      L     L#0;
      U     "MAL1S033Par".Par.FlagProcess.ProcessActive;
      SPBN  n609; // no addition
      SET   ;
      S     "MAL1S033Par".Par.FlagProcess.Inf21; // add heat quantity
      U     "SYS_Scan0_Tick1s"; // scan 1sec
      SPBN  E609;
      L     "MAL1S033Par".Par.ProcessValue_Real.Value05; // heat quantity in kW
      +R    ;
      T     "MAL1S033Par".Par.ProcessValue_Real.Value05;
      SPA   E609;
n609: NOP   0;
      U     "MAL1S033Par".Par.FlagProcess.Inf21; // add heat quantity
      SPBN  E609;
      R     "MAL1S033Par".Par.FlagProcess.Inf21; // add heat quantity
      L     "MAL1S033Par".Par.ProcessValue_Real.Value05;
      L     3.600000e+003;
      /R    ; // from kWs to kWh
      L     1.000000e+003;
      /R    ; // from kWh to MWh
      RND   ;
      T     "MAL1S033Par".Par.ProcessValue_Real.Value06; // result to batch potokoll
      L     0.000000e+000; // clear calculator
      T     "MAL1S033Par".Par.ProcessValue_Real.Value05;
E609: NOP   0;
NETWORK
TITLE =ASW_7000: Step loading kilning
//
      U     "MAL1S033".ToASW.InfDataReady;
      U     "MAL1S033".PCRead.Step.StWait;
      U     "MAL1S033".PCWrite.ExtFuncOn.StartLoading; // PIC command "start loading"
      S     "MAL1S033Par".Par.FlagFunction_1.StepLoading; // Step loading
      R     "MAL1S033Par".Par.FlagMachine.ImpulsNullstellung;
      R     "MAL1S033Par".Par.FlagMachine.CmdTurnRevAfterLoading;
      R     "MAL1S033Par".Par.FlagMachine.CmdTurnFwdAfterLoading;
//
      SET   ;
      R     "MAL1S033".PCWrite.ExtFuncOn.StartLoading; // PIC command "start loading"
//
      U     "MAL1S033".ToASW.InfDataReady;
      U     "MAL1S033".PCRead.Step.StActive;
      U     "MAL1S033Par".Par.FlagFunction_1.StepLoading; // Step loading
      SPB   e71;
      R     "MAL1S033Par".Par.Switches1.StaOn00; // LiftingPositionRound_1
      R     "MAL1S033Par".Par.Switches1.StaOn01; // LiftingPositionRound_2
      R     "MAL1S033Par".Par.Switches1.StaOn02; // LiftingPositionRound_3
      R     "MAL1S033Par".Par.Switches1.StaOn03; // LiftingPositionRound_4
      R     "MAL1S033Par".Par.Switches1.StaOn04; // LiftingPositionRound_5
      R     "MAL1S033Par".Par.Switches1.StaOn05; // LiftingPositionRound_6
e71:  NOP   0;
      U     "MAL1S033".ToASW.InfDataReady;
      U     "MAL1S033".PCRead.Step.StActive;
      U     "MAL1S033Par".Par.FlagFunction_1.StepLoading; // Step loading
      UN    "MAL1S033Par".Par.FlagFunction_1.FinishLoading;
      UN    "MAL1S033Par".Par.FlagFunction_1.LoadEnd;
      SPBN  E700;
      U(    ;
      U(    ;
      L     "G292M".A_3211_MXZ41MA.Ma.OutPositionAngle;
      L     3460; // 346.0°
      >=I   ;
      )     ;
      O     ;
      U(    ;
      L     "G292M".A_3211_MXZ41MA.Ma.OutCntRound;
      L     L#1;
      >=D   ;
      )     ;
      )     ;
      U     "MAL1S033Par".Par.FlagFunction_1.StepLoading;
      =     "MAL1S033Par".Par.FlagFunction_0.ReducedSpeed;
//
      L     "MAL1S033Par".RecipeHeader.Loading.LiftingPositionRound_3;
      L     20; // 20°
      -I    ;
      T     "MAL1S033Par".Par.ParIntMachine.LiftingPositionRound_4;
      L     "MAL1S033Par".RecipeHeader.Loading.LoadingLevelRound_3;
      L     "MAL1S033Par".RecipeHeader.Loading.OffsetLevelNextRound;
      +I    ;
      T     "MAL1S033Par".Par.ParIntMachine.LoadingLevelRound_4;
//
      L     "MAL1S033Par".Par.ParIntMachine.LiftingPositionRound_4;
      L     20; // 20°
      -I    ;
      T     "MAL1S033Par".Par.ParIntMachine.LiftingPositionRound_5;
      L     "MAL1S033Par".Par.ParIntMachine.LoadingLevelRound_4;
      L     "MAL1S033Par".RecipeHeader.Loading.OffsetLevelNextRound;
      +I    ;
      T     "MAL1S033Par".Par.ParIntMachine.LoadingLevelRound_5;
//
      L     "MAL1S033Par".Par.ParIntMachine.LiftingPositionRound_5;
      L     20; // 20°
      -I    ;
      T     "MAL1S033Par".Par.ParIntMachine.LiftingPositionRound_6;
      L     "MAL1S033Par".Par.ParIntMachine.LoadingLevelRound_5;
      L     "MAL1S033Par".RecipeHeader.Loading.OffsetLevelNextRound;
      +I    ;
      T     "MAL1S033Par".Par.ParIntMachine.LoadingLevelRound_6;
//
      L     3600;
      L     "G292M".A_3211_MXZ41MA.Ma.Par.ParTolPosition;
      -I    ;
      L     "G292M".A_3211_MXZ41MA.Ma.OutPositionAngle;
      <=I   ;
      SPB   E700;
//
      L     "G292M".A_3211_MXZ41MA.Ma.OutPositionAngle;
      L     0;
      <I    ;
//      <=I
      SPB   E700;
//
      L     "G292M".A_3211_MXZ41MA.Ma.OutPositionAngle;
      L     10;
      /I    ;
      T     "MAL1S033Par".Par.MachineValue.ISTWERT_FAHRANTRIEB_POSI;
//
      U     "MAL1S033Par".Par.FlagFunction_1.StepLoading; // Step loading
      FP    "MAL1S033Par".Par.Switches1.StaOn08;
      =     "MAL1S033Par".Par.Switches1.StaOn09; // scan start loading
      U     "MAL1S033Par".Par.Switches1.StaOn09; // scan start loading
      SPBN  e72;
      R     "MAL1S033Par".Par.Switches1.StaOn00; // LiftingPositionRound_1
      R     "MAL1S033Par".Par.Switches1.StaOn01; // LiftingPositionRound_2
      R     "MAL1S033Par".Par.Switches1.StaOn02; // LiftingPositionRound_3
      R     "MAL1S033Par".Par.Switches1.StaOn03; // LiftingPositionRound_4
      R     "MAL1S033Par".Par.Switches1.StaOn04; // LiftingPositionRound_5
      R     "MAL1S033Par".Par.Switches1.StaOn05; // LiftingPositionRound_6
//
e72:  NOP   0;
//
      U(    ;
      L     "G292M".A_3211_MXZ41MA.Ma.OutCntRound;
      L     L#0;
      ==D   ;
      )     ;
      U(    ;
      L     "MAL1S033Par".Par.MachineValue.ISTWERT_FAHRANTRIEB_POSI;
      L     "MAL1S033Par".RecipeHeader.Loading.LiftingPositionRound_1;
      <I    ;
      )     ;
      S     "MAL1S033Par".Par.Switches1.StaOn00; // LiftingPositionRound_1
//
      U(    ;
      L     "G292M".A_3211_MXZ41MA.Ma.OutCntRound;
      L     L#0;
      ==D   ;
      )     ;
      U(    ;
      L     "MAL1S033Par".Par.MachineValue.ISTWERT_FAHRANTRIEB_POSI;
      L     "MAL1S033Par".RecipeHeader.Loading.LiftingPositionRound_1;
      >=I   ;
      )     ;
      U(    ;
      L     "MAL1S033Par".Par.MachineValue.ISTWERT_FAHRANTRIEB_POSI;
      L     3550; // 355.0° --> Ruckeln am Nullpunkt abfangen
      <=I   ;
      )     ;
      S     "MAL1S033Par".Par.Switches1.StaOn01; // LiftingPositionRound_2
//
      U     "MAL1S033Par".Par.Switches1.StaOn01; // LiftingPositionRound_2
      R     "MAL1S033Par".Par.Switches1.StaOn00; // LiftingPositionRound_1
//
      U(    ;
      L     "G292M".A_3211_MXZ41MA.Ma.OutCntRound;
      L     L#1;
      ==D   ;
      )     ;
      U(    ;
      L     "MAL1S033Par".Par.MachineValue.ISTWERT_FAHRANTRIEB_POSI;
      L     "MAL1S033Par".RecipeHeader.Loading.LiftingPositionRound_2;
      >=I   ;
      )     ;
      S     "MAL1S033Par".Par.Switches1.StaOn02; // LiftingPositionRound_3
//
      U     "MAL1S033Par".Par.Switches1.StaOn02; // LiftingPositionRound_3
      R     "MAL1S033Par".Par.Switches1.StaOn01; // LiftingPositionRound_2
      R     "MAL1S033Par".Par.Switches1.StaOn00; // LiftingPositionRound_1
//
      U(    ;
      L     "G292M".A_3211_MXZ41MA.Ma.OutCntRound;
      L     L#2;
      ==D   ;
      )     ;
      U(    ;
      L     "MAL1S033Par".Par.MachineValue.ISTWERT_FAHRANTRIEB_POSI;
      L     "MAL1S033Par".RecipeHeader.Loading.LiftingPositionRound_3;
      >=I   ;
      )     ;
      S     "MAL1S033Par".Par.Switches1.StaOn03; // LiftingPositionRound_4
//
      U     "MAL1S033Par".Par.Switches1.StaOn03; // LiftingPositionRound_4
      R     "MAL1S033Par".Par.Switches1.StaOn02; // LiftingPositionRound_3
      R     "MAL1S033Par".Par.Switches1.StaOn01; // LiftingPositionRound_2
      R     "MAL1S033Par".Par.Switches1.StaOn00; // LiftingPositionRound_1
      U(    ;
      L     "G292M".A_3211_MXZ41MA.Ma.OutCntRound;
      L     L#3;
      ==D   ;
      )     ;
      U(    ;
      L     "MAL1S033Par".Par.MachineValue.ISTWERT_FAHRANTRIEB_POSI;
      L     "MAL1S033Par".Par.ParIntMachine.LiftingPositionRound_4;
      >=I   ;
      )     ;
      S     "MAL1S033Par".Par.Switches1.StaOn04; // LiftingPositionRound_5
//
      U     "MAL1S033Par".Par.Switches1.StaOn04; // LiftingPositionRound_5
      R     "MAL1S033Par".Par.Switches1.StaOn03; // LiftingPositionRound_4
      R     "MAL1S033Par".Par.Switches1.StaOn02; // LiftingPositionRound_3
      R     "MAL1S033Par".Par.Switches1.StaOn01; // LiftingPositionRound_2
      R     "MAL1S033Par".Par.Switches1.StaOn00; // LiftingPositionRound_1
      U(    ;
      L     "G292M".A_3211_MXZ41MA.Ma.OutCntRound;
      L     L#4;
      ==D   ;
      )     ;
      U(    ;
      L     "MAL1S033Par".Par.MachineValue.ISTWERT_FAHRANTRIEB_POSI;
      L     "MAL1S033Par".Par.ParIntMachine.LiftingPositionRound_5;
      >=I   ;
      )     ;
      S     "MAL1S033Par".Par.Switches1.StaOn05; // LiftingPositionRound_6
//
      U     "MAL1S033Par".Par.Switches1.StaOn05; // LiftingPositionRound_6
      R     "MAL1S033Par".Par.Switches1.StaOn04; // LiftingPositionRound_5
      R     "MAL1S033Par".Par.Switches1.StaOn03; // LiftingPositionRound_4
      R     "MAL1S033Par".Par.Switches1.StaOn02; // LiftingPositionRound_3
      R     "MAL1S033Par".Par.Switches1.StaOn01; // LiftingPositionRound_2
      R     "MAL1S033Par".Par.Switches1.StaOn00; // LiftingPositionRound_1
      U     "MAL1S033Par".Par.Switches1.StaOn00; // LiftingPositionRound_1
      SPB   Rnd1;
      U     "MAL1S033Par".Par.Switches1.StaOn01; // LiftingPositionRound_2
      SPB   Rnd2;
      U     "MAL1S033Par".Par.Switches1.StaOn02; // LiftingPositionRound_3
      SPB   Rnd3;
      U     "MAL1S033Par".Par.Switches1.StaOn03; // LiftingPositionRound_4
      SPB   Rnd4;
      U     "MAL1S033Par".Par.Switches1.StaOn04; // LiftingPositionRound_5
      SPB   Rnd5;
      U     "MAL1S033Par".Par.Switches1.StaOn05; // LiftingPositionRound_6
      SPB   Rnd6;
      SPA   E700;
Rnd1: NOP   0;
      L     "MAL1S033Par".RecipeHeader.Loading.LoadingLevelRound_1;
      L     "G291M".A_3211_MXZ21_31MA.Ma.Par.ParTolPosition;
      +I    ;
      T     "MAL1S033Par".Par.MachineValue.SOLLWERT_HUBZUG1_HOEHE;
      T     "MAL1S033Par".Par.MachineValue.SOLLWERT_HUBZUG2_HOEHE;
      L     "MAL1S033Par".RecipeHeader.Loading.LoadingSpeed_1;
      T     "MAL1S033Par".Par.MachineValue.SollwertFahrantrieb;
      SPA   E700;
Rnd2: NOP   0;
      L     "MAL1S033Par".RecipeHeader.Loading.LoadingLevelRound_2;
      L     "G291M".A_3211_MXZ21_31MA.Ma.Par.ParTolPosition;
      +I    ;
      T     "MAL1S033Par".Par.MachineValue.SOLLWERT_HUBZUG1_HOEHE;
      T     "MAL1S033Par".Par.MachineValue.SOLLWERT_HUBZUG2_HOEHE;
      L     "MAL1S033Par".RecipeHeader.Loading.LoadingSpeed_2;
      T     "MAL1S033Par".Par.MachineValue.SollwertFahrantrieb;
      SPA   E700;
Rnd3: NOP   0;
      L     "MAL1S033Par".RecipeHeader.Loading.LoadingLevelRound_3;
      L     "G291M".A_3211_MXZ21_31MA.Ma.Par.ParTolPosition;
      +I    ;
      T     "MAL1S033Par".Par.MachineValue.SOLLWERT_HUBZUG1_HOEHE;
      T     "MAL1S033Par".Par.MachineValue.SOLLWERT_HUBZUG2_HOEHE;
      L     "MAL1S033Par".RecipeHeader.Loading.LoadingSpeed_3;
      T     "MAL1S033Par".Par.MachineValue.SollwertFahrantrieb;
      SPA   E700;
Rnd4: NOP   0;
      L     "MAL1S033Par".Par.ParIntMachine.LoadingLevelRound_4;
      L     "G291M".A_3211_MXZ21_31MA.Ma.Par.ParTolPosition;
      +I    ;
      T     "MAL1S033Par".Par.MachineValue.SOLLWERT_HUBZUG1_HOEHE;
      T     "MAL1S033Par".Par.MachineValue.SOLLWERT_HUBZUG2_HOEHE;
//      L     "MAL1S033Par".RecipeHeader.Loading.LoadingSpeed_3
      L     87; // 87%
      T     "MAL1S033Par".Par.MachineValue.SollwertFahrantrieb;
      SPA   E700;
Rnd5: NOP   0;
      L     "MAL1S033Par".Par.ParIntMachine.LoadingLevelRound_5;
      L     "G291M".A_3211_MXZ21_31MA.Ma.Par.ParTolPosition;
      +I    ;
      T     "MAL1S033Par".Par.MachineValue.SOLLWERT_HUBZUG1_HOEHE;
      T     "MAL1S033Par".Par.MachineValue.SOLLWERT_HUBZUG2_HOEHE;
//      L     "MAL1S033Par".RecipeHeader.Loading.LoadingSpeed_3
      L     87; // 87%
      T     "MAL1S033Par".Par.MachineValue.SollwertFahrantrieb;
      SPA   E700;
Rnd6: NOP   0;
      L     "MAL1S033Par".Par.ParIntMachine.LoadingLevelRound_6;
      L     "G291M".A_3211_MXZ21_31MA.Ma.Par.ParTolPosition;
      +I    ;
      T     "MAL1S033Par".Par.MachineValue.SOLLWERT_HUBZUG1_HOEHE;
      T     "MAL1S033Par".Par.MachineValue.SOLLWERT_HUBZUG2_HOEHE;
//      L     "MAL1S033Par".RecipeHeader.Loading.LoadingSpeed_3
      L     87; // 87%
      T     "MAL1S033Par".Par.MachineValue.SollwertFahrantrieb;
      SPA   E700;
E700: NOP   0;
NETWORK
TITLE =Sub 7010: Kilning  loading finished
//      L     0;
//      L     "MAL1S033".ToSSW.InPrevSecDB;
//      ==I   ;
//      SPB   fin;
//      O(;
//      U     "MAL1S017Par".Par.FlagFunction_1.FinishUnloading;
//      U     "MAL1S033".PCWrite.ExtFuncOn.FinishLoading; // PIC command "finish
//loading"
//      O       "MAL1S017Par".Par.FlagFunction_1.StepCleaning;
//      U     "MAL1S017".PCRead.Step.StEmptied;
//      U(    ;
//      AUF   "MAL1S017";
//      L DBNO;
//      L     "MAL1S033".ToSSW.InPrevSecDB;
//      ==I;
//      )     ;
//      )     ;
//      O(;
//      U     "MAL1S018Par".Par.FlagFunction_1.FinishUnloading;
//      U     "MAL1S033".PCWrite.ExtFuncOn.FinishLoading; // PIC command "finish
//loading"
//      O       "MAL1S018Par".Par.FlagFunction_1.StepCleaning;
//      U     "MAL1S018".PCRead.Step.StEmptied;
//      U(    ;
//      AUF   "MAL1S018";
//      L DBNO;
//      L     "MAL1S033".ToSSW.InPrevSecDB;
//      ==I;
//      )     ;
//      )     ;
//      O(;
//      U     "MAL1S019Par".Par.FlagFunction_1.FinishUnloading;
//      U     "MAL1S033".PCWrite.ExtFuncOn.FinishLoading; // PIC command "finish
//loading"
//      O       "MAL1S019Par".Par.FlagFunction_1.StepCleaning;
//      U     "MAL1S019".PCRead.Step.StEmptied;
//      U(    ;
//      AUF   "MAL1S019";
//      L DBNO;
//      L     "MAL1S033".ToSSW.InPrevSecDB;
//      ==I;
//      )     ;
//      )     ;
//      O(;
//      U     "MAL1S020Par".Par.FlagFunction_1.FinishUnloading;
//      U     "MAL1S033".PCWrite.ExtFuncOn.FinishLoading; // PIC command "finish
//loading"
//      O       "MAL1S020Par".Par.FlagFunction_1.StepCleaning;
//      U     "MAL1S020".PCRead.Step.StEmptied;
//      U(    ;
//      AUF   "MAL1S020";
//      L DBNO;
//      L     "MAL1S033".ToSSW.InPrevSecDB;
//      ==I;
//      )     ;
//      )     ;
//      O(;
//      U     "MAL1S021Par".Par.FlagFunction_1.FinishUnloading;
//      U     "MAL1S033".PCWrite.ExtFuncOn.FinishLoading; // PIC command "finish
//loading"
//      O       "MAL1S021Par".Par.FlagFunction_1.StepCleaning;
//      U     "MAL1S021".PCRead.Step.StEmptied;
//      U(    ;
//      AUF   "MAL1S021";
//      L DBNO;
//      L     "MAL1S033".ToSSW.InPrevSecDB;
//      ==I;
//      )     ;
//      )     ;
//      O(;
//      U     "MAL1S022Par".Par.FlagFunction_1.FinishUnloading;
//      U     "MAL1S033".PCWrite.ExtFuncOn.FinishLoading; // PIC command "finish
//loading"
//      O       "MAL1S022Par".Par.FlagFunction_1.StepCleaning;
//      U     "MAL1S022".PCRead.Step.StEmptied;
//      U(    ;
//      AUF   "MAL1S022";
//      L DBNO;
//      L     "MAL1S033".ToSSW.InPrevSecDB;
//      ==I;
//      )     ;
//      )     ;
//      O(;
//      U     "MAL1S023Par".Par.FlagFunction_1.FinishUnloading;
//      U     "MAL1S033".PCWrite.ExtFuncOn.FinishLoading; // PIC command "finish l
//oading"
//      O       "MAL1S023Par".Par.FlagFunction_1.StepCleaning;
//      U     "MAL1S023".PCRead.Step.StEmptied;
//      U(    ;
//      AUF   "MAL1S023";
//      L DBNO;
//      L     "MAL1S033".ToSSW.InPrevSecDB;
//      ==I;
//      )     ;
//      )     ;
//      O(;
//      U     "MAL1S024Par".Par.FlagFunction_1.FinishUnloading;
//      U     "MAL1S033".PCWrite.ExtFuncOn.FinishLoading; // PIC command "finish
//loading"
//      O       "MAL1S024Par".Par.FlagFunction_1.StepCleaning;
//      U     "MAL1S024".PCRead.Step.StEmptied;
//      U(    ;
//      AUF   "MAL1S024";
//      L DBNO;
//      L     "MAL1S033".ToSSW.InPrevSecDB;
//      ==I;
//      )     ;
//      )     ;
//      O(    ;
//      U     "MAL1S033Par".Par.FlagFunction_1.StepLoading; // Step loading
//      UN    "MAL1S033".ToASW.InfSameJobPrevSec;
//      U     "MAL1S033".PCWrite.ExtFuncOn.FinishLoading; // PIC command "finish l
//oading"
//      )     ;
//      U     "MAL1S033".ToASW.InfDataReady;
//      U     "MAL1S033".PCRead.Step.StActive;
//      S     "MAL1S033Par".Par.FlagFunction_1.LoadEnd;
////
//      U     "MAL1S033".PCWrite.ExtFuncOn.FinishLoading; // PIC command "finish
//loading"
//      R     "MAL1S033".PCWrite.ExtFuncOn.FinishLoading; // PIC command "finish l
//oading"
////
//      U     "MAL1S033Par".Par.FlagFunction_1.LoadEnd;
//      U     "MAL1S033Par".Par.FlagFunction_1.StepLoading; // Step loading
//      FP    "MAL1S033Par".Par.FlagFunction_0.ImpulsSollposition;
//      =     "MAL1S033Par".Par.FlagFunction_0.MerkerSollpositionFP;
//      U     "MAL1S033Par".Par.FlagFunction_0.MerkerSollpositionFP;
//      SPBN  fin;
//      L     WinCoS_BIW01_09PLC1BIW01_02.Ma.OutPositionAngle;
//      L     "MAL1S033Par".Par.ParIntProcess.LoadingOverlap;
//      +I    ;
//      T     WinCoS_BIW01_09PLC1BIW01_02.Ma.InPositionTarget;
////???      SET
////???      S     "PLC1BIW01_02".TurningTo_Parkposition    //
//WinCoS_BIW01_09PLC1BIW01_02..Ma.InAdjusting
//// Beladehöhe speichern
//      L     "MAL1S033Par".Par.MachineValue.SOLLWERT_HUBZUG1_HOEHE;
//      T     "MAL1S033Par".Par.ParIntMachine.LastLoadingLevel; // saved loading
//value
//fin:  NOP   0;
//E701: NOP   0;
// Grundschicht vollständig bedeckt
      U(    ;
// Die Position bei IBN ermitteln!
      L     "G292M".A_3211_MXZ41MA.Ma.OutPositionAngle;
      L     3564; // 356.4°
      >=I   ;
      )     ;
      U     "MAL1S033Par".Par.FlagFunction_1.StepLoading;
      U     "G292M".A_3211_MXZ41MA.Ma.InEnableFwd;
      S     "MAL1S033Par".Par.FlagFunction_1.LoadFirstPartEnd;
      S     "MAL1S033Par".Par.FlagProcess.Product_Inside;

      U     "MAL1S033Par".Par.FlagProcess.ProcessActive;
      U     "MAL1S033Par".Par.FlagFunction_1.FinishLoading;
      O     "MAL1S033Par".Par.FlagFunction_1.StepUnloading;
      O     "MAL1S033".PCRead.Step.StIdling; // "SecDB".PCRead.Step.StIdling
      R     "MAL1S033Par".Par.FlagFunction_1.LoadFirstPartEnd;

      L     0;
      L     "MAL1S033".ToSSW.InPrevSecDB;
      ==I   ;
      SPB   fin;
      O(    ;
      U     "MAL1S017Par".Par.FlagFunction_1.FinishUnloading;
      U     "MAL1S017".PCWrite.ExtFuncOn.FinishCleanSurface; // PIC command "finish unloading"
//      U       "MAL1S033".PCWrite.ExtFuncOn.FinishLoading    // PIC command "finish loading"
      O     "MAL1S017Par".Par.FlagFunction_1.StepCleaning;
      U     "MAL1S017".PCRead.Step.StEmptied;
      U(    ;
      AUF   "MAL1S017";
      L     DBNO;
      L     "MAL1S033".ToSSW.InPrevSecDB;
      ==I   ;
      )     ;
      )     ;
      O(    ;
      U     "MAL1S018Par".Par.FlagFunction_1.FinishUnloading;
      U     "MAL1S018".PCWrite.ExtFuncOn.FinishCleanSurface; // PIC command "finish unloading"
//      U       "MAL1S033".PCWrite.ExtFuncOn.FinishLoading    // PIC command "finish loading"
      O     "MAL1S018Par".Par.FlagFunction_1.StepCleaning;
      U     "MAL1S018".PCRead.Step.StEmptied;
      U(    ;
      AUF   "MAL1S018";
      L     DBNO;
      L     "MAL1S033".ToSSW.InPrevSecDB;
      ==I   ;
      )     ;
      )     ;
      O(    ;
      U     "MAL1S019Par".Par.FlagFunction_1.FinishUnloading;
      U     "MAL1S019".PCWrite.ExtFuncOn.FinishCleanSurface; // PIC command "finish unloading"
//      U       "MAL1S033".PCWrite.ExtFuncOn.FinishLoading    // PIC command "finish loading"
      O     "MAL1S019Par".Par.FlagFunction_1.StepCleaning;
      U     "MAL1S019".PCRead.Step.StEmptied;
      U(    ;
      AUF   "MAL1S019";
      L     DBNO;
      L     "MAL1S033".ToSSW.InPrevSecDB;
      ==I   ;
      )     ;
      )     ;
      O(    ;
      U     "MAL1S020Par".Par.FlagFunction_1.FinishUnloading;
      U     "MAL1S020".PCWrite.ExtFuncOn.FinishCleanSurface; // PIC command "finish unloading"
//      U       "MAL1S033".PCWrite.ExtFuncOn.FinishLoading    // PIC command "finish loading"
      O     "MAL1S020Par".Par.FlagFunction_1.StepCleaning;
      U     "MAL1S020".PCRead.Step.StEmptied;
      U(    ;
      AUF   "MAL1S020";
      L     DBNO;
      L     "MAL1S033".ToSSW.InPrevSecDB;
      ==I   ;
      )     ;
      )     ;
      O(    ;
      U     "MAL1S021Par".Par.FlagFunction_1.FinishUnloading;
      U     "MAL1S021".PCWrite.ExtFuncOn.FinishCleanSurface; // PIC command "finish unloading"
//      U       "MAL1S033".PCWrite.ExtFuncOn.FinishLoading    // PIC command "finish loading"
      O     "MAL1S021Par".Par.FlagFunction_1.StepCleaning;
      U     "MAL1S021".PCRead.Step.StEmptied;
      U(    ;
      AUF   "MAL1S021";
      L     DBNO;
      L     "MAL1S033".ToSSW.InPrevSecDB;
      ==I   ;
      )     ;
      )     ;
      O(    ;
      U     "MAL1S022Par".Par.FlagFunction_1.FinishUnloading;
      U     "MAL1S022".PCWrite.ExtFuncOn.FinishCleanSurface; // PIC command "finish unloading"
//      U       "MAL1S033".PCWrite.ExtFuncOn.FinishLoading    // PIC command "finish loading"
      O     "MAL1S022Par".Par.FlagFunction_1.StepCleaning;
      U     "MAL1S022".PCRead.Step.StEmptied;
      U(    ;
      AUF   "MAL1S022";
      L     DBNO;
      L     "MAL1S033".ToSSW.InPrevSecDB;
      ==I   ;
      )     ;
      )     ;
      O(    ;
      U     "MAL1S023Par".Par.FlagFunction_1.FinishUnloading;
      U     "MAL1S023".PCWrite.ExtFuncOn.FinishCleanSurface; // PIC command "finish unloading"
//      U       "MAL1S033".PCWrite.ExtFuncOn.FinishLoading    // PIC command "finish loading"
      O     "MAL1S033Par".Par.FlagFunction_1.StepCleaning;
      U     "MAL1S033".PCRead.Step.StEmptied;
      U(    ;
      AUF   "MAL1S023";
      L     DBNO;
      L     "MAL1S023".ToSSW.InPrevSecDB;
      ==I   ;
      )     ;
      )     ;
      O(    ;
      U     "MAL1S024Par".Par.FlagFunction_1.FinishUnloading;
      U     "MAL1S024".PCWrite.ExtFuncOn.FinishCleanSurface; // PIC command "finish unloading"
//      U       "MAL1S033".PCWrite.ExtFuncOn.FinishLoading    // PIC command "finish loading"
      O     "MAL1S024Par".Par.FlagFunction_1.StepCleaning;
      U     "MAL1S024".PCRead.Step.StEmptied;
      U(    ;
      AUF   "MAL1S024";
      L     DBNO;
      L     "MAL1S033".ToSSW.InPrevSecDB;
      ==I   ;
      )     ;
      )     ;
//      O(
//      U       "MAL1S033Par".Par.FlagFunction_1.StepLoading    // Step loading
//      UN      "MAL1S033".ToASW.InfSameJobPrevSec
//      U       "MAL1S033".PCWrite.ExtFuncOn.FinishLoading    // PIC command "finish loading"
//      )
      U     "MAL1S033".ToASW.InfDataReady;
      U     "MAL1S033".PCRead.Step.StActive;
      U     "MAL1S033Par".Par.FlagFunction_1.LoadFirstPartEnd;
      S     "MAL1S033Par".Par.FlagFunction_1.LoadEnd;
      R     "MAL1S017".PCWrite.ExtFuncOn.FinishCleanSurface; // PIC command "finish unloading"
      R     "MAL1S018".PCWrite.ExtFuncOn.FinishCleanSurface; // PIC command "finish unloading"
      R     "MAL1S019".PCWrite.ExtFuncOn.FinishCleanSurface; // PIC command "finish unloading"
      R     "MAL1S020".PCWrite.ExtFuncOn.FinishCleanSurface; // PIC command "finish unloading"
      R     "MAL1S021".PCWrite.ExtFuncOn.FinishCleanSurface; // PIC command "finish unloading"
      R     "MAL1S022".PCWrite.ExtFuncOn.FinishCleanSurface; // PIC command "finish unloading"
      R     "MAL1S023".PCWrite.ExtFuncOn.FinishCleanSurface; // PIC command "finish unloading"
      R     "MAL1S024".PCWrite.ExtFuncOn.FinishCleanSurface; // PIC command "finish unloading"

//
      U     "MAL1S033".PCWrite.ExtFuncOn.FinishLoading; // PIC command "finish loading"
      R     "MAL1S033".PCWrite.ExtFuncOn.FinishLoading; // PIC command "finish loading"
//
      U     "MAL1S033Par".Par.FlagFunction_1.LoadEnd;
      U     "MAL1S033Par".Par.FlagFunction_1.StepLoading; // Step loading
      FP    "MAL1S033Par".Par.FlagFunction_0.ImpulsSollposition;
      =     "MAL1S033Par".Par.FlagFunction_0.MerkerSollpositionFP;
      U     "MAL1S033Par".Par.FlagFunction_0.MerkerSollpositionFP;
      SPBN  fin;
      L     "G292M".A_3211_MXZ41MA.Ma.OutPositionAngle;
      L     "MAL1S033Par".Par.ParIntProcess.LoadingOverlap;
      +I    ;
      T     "G292M".A_3211_MXZ41MA.Ma.InPositionTarget;
      SET   ;
      S     "G292M".TurningTo_Parkposition;

// Extra Planierrunde wenn der Fahrantrieb ueber 346° beim Beladen Ende war
      L     "G292M".A_3211_MXZ41MA.Ma.OutPositionAngle;
      L     3460; // 346,0 °
      >I    ;
      S     "G292M".Turning_One_Round_More;

// Beladehöhe speichern
      L     "MAL1S033Par".Par.MachineValue.SOLLWERT_HUBZUG1_HOEHE;
      T     "MAL1S033Par".Par.ParIntMachine.LastLoadingLevel; // saved loading value
fin:  NOP   0;

// Hubzüge erst auf der Parkposition abheben
      U     "G292M".TurningTo_Parkposition;
      FN    "G291M".USW8;
      =     "G291M".USW9;

      U     "G291M".USW9;
      O     ;
      U     "MAL1S033Par".Par.FlagFunction_1.FinishLoading;
      U(    ;
      U     "G292M".A_3211_MXZ41MA.A_3211_BZS43.StCtoTrue; // sensor zero point
      O     "G292M".A_3211_MXZ41MA.A_3211_BZS43.StTrue; // sensor zero point
      )     ;
      SPBN  auf;
      L     "G291M".A_3211_MXZ21_31MA.Ma.Par.ParPositionTopLeftUnits; //LIFTING DRIVE
      L     150;
      +I    ;
      T     "MAL1S033Par".Par.MachineValue.SOLLWERT_HUBZUG1_HOEHE;
      L     "G291M".A_3211_MXZ21_31MA.Ma.Par.ParPositionTopRightUnits; //LIFTING DRIVE
      L     150;
      +I    ;
      T     "MAL1S033Par".Par.MachineValue.SOLLWERT_HUBZUG2_HOEHE;
      L     1;
      T     "G291M".A_3211_MXZ21_31MA.Ma.Par.ParTolPosition;
auf:  NOP   0;

      NOP   0;
NETWORK
TITLE =ASW_6080: Processtime Kilning
//      CALL  "SSA_MH_ProcessTime_Fct" , DB1017
//       InfDataReady :="MAL1S017".ToASW.InfDataReady
//       ProzessActive:="MAL1S017Par".Par.FlagProcess.ProcessActive
//       InStartTime  :="MAL1S017Par".Prozesstime.Starttime
//       OutStartTime :="MAL1S017Par".Prozesstime.Starttime
//       ProcessTime  :="MAL1S017Par".Prozesstime
//
      CALL "SSA_MH_ProcessTime_Fct" , DB  1033 (
           InfDataReady             := "MAL1S033".ToASW.InfDataReady,
           ProzessActive            := "MAL1S033Par".Par.FlagProcess.ProcessActive,
           InStartTime              := "MAL1S033Par".Processtime.StartTime,
           OutStartTime             := "MAL1S033Par".Processtime.StartTime,
           ProcessTime              := "MAL1S033Par".Processtime);

NETWORK
TITLE =Sub 7020: Step start process kilning

      U     "MAL1S033".ToASW.InfDataReady;
      U     "MAL1S033".PCRead.Step.StActive;
//      U       "MAL1S033".PCWrite.ExtFuncOn.StartProcess    // PIC command "start process kilning"
      U     "MAL1S033Par".Par.FlagFunction_1.LoadEnd;

      U     "G292M".A_3211_MXZ41MA.A_3211_BZS43.StTrue; // sensor zero point
      U     "G291M".A_3211_MXZ21_31MA.A_3211_BZS23.InpTrue;
      U     "G291M".A_3211_MXZ21_31MA.A_3211_BZS33.InpTrue;

      O(    ;
      UN    "MAL1S033".SecNom.Par1On.Cmd01; // With Loading
      UN    "MAL1S033".ToASW.InfSameBatchPrevSec;
      U     "MAL1S033".ToASW.InfDataReady;
      U     "MAL1S033".PCRead.Step.StActive;
      )     ;

      S     "MAL1S033Par".Par.FlagFunction_1.FinishLoading; // start process kilning
      R     "MAL1S033Par".Par.FlagFunction_1.LoadEnd;
//
      U     "MAL1S033".PCWrite.ExtFuncOn.StartProcess; // PIC command "start process kilning"
      R     "MAL1S033".PCWrite.ExtFuncOn.StartProcess; // PIC command "start process kilning"
//
      U     "G292M".A_3211_MXZ41MA.Ma.StAdjusted;
      O     "G292M".A_3211_MXZ41MA.Ma.OutAdjusted;
      U     "MAL1S033Par".Par.FlagFunction_1.FinishLoading; // start process kilning
      O     "MAL1S033Par".Par.FlagProcess.ProcessActive;
      SPBN  E702;
      L     "G291M".A_3211_MXZ21_31MA.Ma.Par.ParPositionTopLeftUnits; //LIFTING DRIVE
      L     50; //jk
      +I    ;
      T     "MAL1S033Par".Par.MachineValue.SOLLWERT_HUBZUG1_HOEHE;
      L     "G291M".A_3211_MXZ21_31MA.Ma.Par.ParPositionTopRightUnits; //LIFTING DRIVE
      L     50; //jk
      +I    ;
      T     "MAL1S033Par".Par.MachineValue.SOLLWERT_HUBZUG2_HOEHE;
      L     1;
      T     "G291M".A_3211_MXZ21_31MA.Ma.Par.ParTolPosition;

E702: NOP   0;

      U     "G292M".TurningTo_Parkposition;
      SPBN  E703;
      U(    ;
      L     "G292M".A_3211_MXZ41MA.Ma.OutPositionAngle;
      L     3500;
      >=I   ;
      )     ;
      SPBN  E703;
      L     10; // 10% speed to parkposition
      T     "MAL1S033Par".Par.MachineValue.SollwertFahrantrieb;
E703: NOP   0;

      U     "G292M".TurningTo_Parkposition;
      SPBN  E704;
      U(    ;
      L     "G292M".A_3211_MXZ41MA.Ma.OutPositionAngle;
      L     3500;
      <I    ;
      )     ;
      SPBN  E704;
      L     87; // 87% speed to parkposition
      T     "MAL1S033Par".Par.MachineValue.SollwertFahrantrieb;
E704: NOP   0;

NETWORK
TITLE =ASW_8000:  Step unloading kilning

      UN    "MAL1S033Par".Par.FlagFunction_1.StepUnloading; // Step Unloading
      R     "MAL1S033Par".Par.FlagFunction_0.OverlapSaved; // Ueberlappung erfasst
//
      U     "MAL1S033".ToASW.InfDataReady;
      U     "MAL1S033".PCRead.Step.StEmptying;
      U(    ;
      L     "MAL1S033Par".RecipeHeader.Unloading.StartUnloadAuto; //StartUnloadAuto = 0
      L     1;
      <>I   ;
      U     "MAL1S033".PCWrite.ExtFuncOn.StartUnLoading; // PIC command "start unloading"
      O     ;
      U(    ;
      L     "MAL1S033Par".RecipeHeader.Unloading.StartUnloadAuto; //StartUnloadAuto = 10
      L     1;
      ==I   ;
      )     ;
      UN    "G297M".A_3225_TSC01_AF.OutL; // 30% Ventilatordrehzahl
      UN    "G297M".A_3226_TSC01_AF.OutL; // 30% Ventilatordrehzahl
      )     ;
      S     "MAL1S033Par".Par.FlagFunction_1.StepUnloading; // Step Unloading
      R     "MAL1S033Par".Par.FlagMachine.ImpulsNullstellung;
      R     "MAL1S023Par".Par.FlagMachine.WEGMESSUNG_0;
      R     DB923.DBX  148.0; // FP
      R     "MAL1S033Par".Par.FlagMachine.CmdTurnRevAfterUnloading;
      R     "MAL1S033Par".Par.FlagMachine.CmdTurnFwdAfterUnloading;
//
      SET   ;
      R     "MAL1S033".PCWrite.ExtFuncOn.StartUnLoading; // PIC command "start unloading"
//
      U     "MAL1S033".ToASW.InfDataReady;
      U     "MAL1S033".PCRead.Step.StEmptying;
      U     "MAL1S033Par".Par.FlagFunction_1.StepUnloading; // Step Unloading
      SPBN  e800;
      L     "MAL1S033Par".Par.ParIntMachine.LastLoadingLevel; // saved loading value
      T     "MAL1S033Par".Par.ParIntMachine.FUELLHOEHE_PRODUKT;
//
      U(    ;
      L     "G291M".A_3211_MXZ21_31MA.Ma.OutPositionLeft;
      L     "MAL1S033Par".Par.ParIntMachine.FUELLHOEHE_PRODUKT;
      >I    ;
      )     ;
      O(    ;
      L     "G291M".A_3211_MXZ21_31MA.Ma.OutPositionRight;
      L     "MAL1S033Par".Par.ParIntMachine.FUELLHOEHE_PRODUKT;
      >I    ;
      )     ;
      UN(   ;
      U(    ;
      L     "G291M".A_3211_MXZ21_31MA.Ma.OutPositionLeft;
      L     "MAL1S033Par".Par.MachineValue.SOLLWERT_HUBZUG1_HOEHE;
      <=I   ;
      )     ;
      U(    ;
      L     "G291M".A_3211_MXZ21_31MA.Ma.OutPositionRight;
      L     "MAL1S033Par".Par.MachineValue.SOLLWERT_HUBZUG1_HOEHE;
      <=I   ;
      )     ;
      )     ;
      =     "MAL1S033Par".Par.FlagFunction_0.ScrewAboveProductLayer; // HubzuegeUeberProdukt
//
//- Letzte Entladehoehe erreicht ---
      U(    ;
      L     "MAL1S033Par".Par.MachineValue.SOLLWERT_HUBZUG1_HOEHE;
      L     0;
      <=I   ;
      )     ;
      U(    ;
      L     "MAL1S033Par".Par.MachineValue.SOLLWERT_HUBZUG1_HOEHE;
      L     "G291M".A_3211_MXZ21_31MA.Ma.InPositionTarget;
      ==I   ;
      )     ;
      U     "G291M".A_3211_MXZ21_31MA.Ma.StAdjusted;
      U     "MAL1S033Par".Par.FlagFunction_1.StepUnloading; // Step Unloading
      FP    "MAL1S033Par".Par.FlagFunction_0.UnloadLevelReachedFP; // UnloadLevelReachedFP
      =     "MAL1S033Par".Par.FlagFunction_0.ImpulsUnloadLevelReached; // ImpulsUnloadLevelReached
      UN    "MAL1S033Par".Par.FlagFunction_0.ImpulsUnloadLevelReached; // ImpulsUnloadLevelReached
      O     "MAL1S033Par".Par.FlagFunction_0.OverlapSaved; // Ueberlappung erfasst
      SPB   over;
      L     "G292M".A_3211_MXZ41MA.Ma.OutCntRound;
      L     1;
      +I    ;
      T     "MAL1S033Par".Par.ParIntProcess.UnloadungRounds;
//
      L     "G292M".A_3211_MXZ41MA.Ma.OutPositionAngle;
      L     3600; // 360,0°
      >=I   ;
      SPBN  soz1;
      -I    ;
      SPA   soz2;
soz1: NOP   0;
      TAK   ;
soz2: NOP   0;
      L     100; // 10,0°
      +I    ;
      T     "MAL1S033Par".Par.ParIntProcess.UnloadingOverlap;
      T     "G292M".A_3211_MXZ41MA.Ma.InPositionTarget;
      S     "MAL1S033Par".Par.FlagFunction_0.OverlapSaved; // Ueberlappung erfasst
over: NOP   0;
      U(    ;
      L     "G292M".A_3211_MXZ41MA.Ma.OutCntRound;
      L     L#0;
      ==D   ;
      )     ;
      SPB   rnd1;
      L     "G292M".A_3211_MXZ41MA.Ma.OutCntRound;
      L     L#1;
      ==D   ;
      SPB   rnd2;
      L     "G292M".A_3211_MXZ41MA.Ma.OutCntRound;
      L     L#2;
      >=D   ;
      SPB   rnd3;
      SPA   e801;
rnd1: NOP   0;
      L     "MAL1S033Par".RecipeHeader.Loading.LiftingPositionRound_3;
      T     "MAL1S033Par".Par.MachineValue.SOLLWERT_HUBZUG1_HOEHE;
      T     "MAL1S033Par".Par.MachineValue.SOLLWERT_HUBZUG2_HOEHE;
      L     1;
      T     "G291M".A_3211_MXZ21_31MA.Ma.Par.ParTolPosition;
      L     "MAL1S033Par".RecipeHeader.Unloading.UnLoadingSpeed_1;
      T     "MAL1S033Par".Par.MachineValue.SollwertFahrantrieb;
      SPA   e801;
rnd2: NOP   0;
      L     "MAL1S033Par".RecipeHeader.Loading.LiftingPositionRound_4;
      T     "MAL1S033Par".Par.MachineValue.SOLLWERT_HUBZUG1_HOEHE;
      T     "MAL1S033Par".Par.MachineValue.SOLLWERT_HUBZUG2_HOEHE;
      L     1;
      T     "G291M".A_3211_MXZ21_31MA.Ma.Par.ParTolPosition;
      L     "MAL1S033Par".RecipeHeader.Unloading.UnLoadingSpeed_2;
      T     "MAL1S033Par".Par.MachineValue.SollwertFahrantrieb;
      SPA   e801;
rnd3: NOP   0;
      L     "MAL1S033Par".RecipeHeader.Loading.LiftingPositionRound_5;
      T     "MAL1S033Par".Par.MachineValue.SOLLWERT_HUBZUG1_HOEHE;
      T     "MAL1S033Par".Par.MachineValue.SOLLWERT_HUBZUG2_HOEHE;
      L     1;
      T     "G291M".A_3211_MXZ21_31MA.Ma.Par.ParTolPosition;
      L     "MAL1S033Par".RecipeHeader.Unloading.UnLoadingSpeed_3;
      T     "MAL1S033Par".Par.MachineValue.SollwertFahrantrieb;
      SPA   e801;

e801: NOP   0;
      U     "MAL1S033".ToASW.InfDataReady;
      U     "MAL1S033".PCRead.Step.StEmptying;
      U     "MAL1S033Par".Par.FlagFunction_1.StepUnloading; // Step Unloading
      U(    ;
      L     "G292M".A_3211_MXZ41MA.Ma.OutCntRound;
      L     "MAL1S033Par".Par.ParIntProcess.UnloadungRounds;
      >=I   ;
      )     ;
      U     "G291M".A_3211_MXZ21_31MA.Ma.StAdjusted;
      U     "G292M".A_3211_MXZ41MA.Ma.StAdjusted;
      S     "MAL1S033Par".Par.FlagFunction_1.FinishUnloading;

      U     "MAL1S033".ToASW.InfDataReady;
      U     "MAL1S033".PCRead.Step.StEmptying;
      U     "MAL1S033Par".Par.FlagFunction_1.FinishUnloading;
      SPBN  e800;
      L     "G291M".A_3211_MXZ21_31MA.Ma.Par.ParPositionTopLeftUnits;
      L     50;
      +I    ;
      T     "MAL1S033Par".Par.MachineValue.SOLLWERT_HUBZUG1_HOEHE;
      L     "G291M".A_3211_MXZ21_31MA.Ma.Par.ParPositionTopRightUnits;
      L     50;
      +I    ;
      T     "MAL1S033Par".Par.MachineValue.SOLLWERT_HUBZUG2_HOEHE;
      L     1;
      T     "G291M".A_3211_MXZ21_31MA.Ma.Par.ParTolPosition;

      L     0;
      T     "MAL1S033Par".Par.ParIntMachine.LastLoadingLevel; // saved loading value
      T     "MAL1S033Par".Par.ParIntMachine.FUELLHOEHE_PRODUKT;
e800: NOP   0;
//
// --> Wie bei der Bank Avangard
      U     "MAL1S033Par".Par.FlagFunction_1.StepUnloading;
      U     "MAL1S033Par".Par.FlagFunction_1.FinishUnloading;
      FP    DB923.DBX  148.0;
      =     DB923.DBX  148.1;
      SPBN  TAU1;
      L     "G292M".A_3211_MXZ41MA.Ma.OutPositionAngle;
      L     1800;
      <I    ;
      S     "MAL1S033Par".Par.FlagMachine.CmdTurnRevAfterUnloading;
      L     "G292M".A_3211_MXZ41MA.Ma.OutPositionAngle;
      L     1800;
      >=I   ;
      S     "MAL1S033Par".Par.FlagMachine.CmdTurnFwdAfterUnloading;
TAU1: NOP   0;
      U     "MAL1S033Par".Par.FlagMachine.CmdTurnRevAfterUnloading;
      O     "MAL1S033Par".Par.FlagMachine.CmdTurnFwdAfterUnloading;
      U     "MAL1S033Par".Par.FlagFunction_1.FinishUnloading;
      U     "G293M".A_3211_MXZ11.StStopped;
      U     "G291M".A_3211_MXZ21_31MA.Ma.OutHigherMinPos;
      U(    ;
      U     "G291M".A_3211_MXZ21_31MA.A_3211_BZS33.InpTrue;
      U     "G291M".A_3211_MXZ21_31MA.A_3211_BZS23.InpTrue;
      O     "G291M".A_3211_MXZ21_31MA.Ma.StAdjusted;
      )     ;
      S     "MAL1S033Par".Par.FlagMachine.WEGMESSUNG_0;
//
      U     "MAL1S033".ToASW.InfDataReady;
      U     "MAL1S033Par".Par.FlagFunction_1.FinishUnloading;
      U     "MAL1S033Par".Par.FlagMachine.WEGMESSUNG_0;
      SPBN  TAU2;
//    L       "MAL1S033Par".RecipeHeader.Cleaning.CleaningSpeed_1
      L     30; // 30%
      T     "MAL1S033Par".Par.MachineValue.SollwertFahrantrieb;
TAU2: NOP   0;
      NOP   0;
NETWORK
TITLE =ASW_9000: Step cleaning
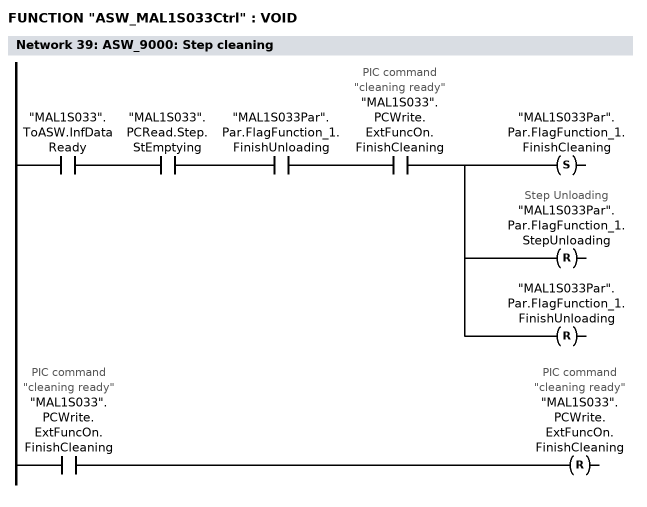

      U     "MAL1S033".ToASW.InfDataReady;
      U     "MAL1S033".PCRead.Step.StEmptying;
      U     "MAL1S033Par".Par.FlagFunction_1.FinishUnloading;
      U     "MAL1S033".PCWrite.ExtFuncOn.FinishCleaning; // PIC command "cleaning ready"
      S     "MAL1S033Par".Par.FlagFunction_1.FinishCleaning;
      R     "MAL1S033Par".Par.FlagFunction_1.StepUnloading; // Step Unloading
      R     "MAL1S033Par".Par.FlagFunction_1.FinishUnloading;
//
      U     "MAL1S033".PCWrite.ExtFuncOn.FinishCleaning; // PIC command "cleaning ready"
      R     "MAL1S033".PCWrite.ExtFuncOn.FinishCleaning; // PIC command "cleaning ready"
NETWORK
TITLE =ASW_9080: Send section date to PIC after germination

      AUF   "MAL1S033";
      U     "MAL1S033".PCRead.Step.StEmptying;
      FP    "MAL1S033Par".Par.FlagProcess.FP_SendResultToPIC;
      SPBN  E908;
//

E908: NOP   0;
NETWORK
TITLE =ASW_10000: ILO functions

      U     "MAL1S033".SecAc.Sta1On.Inf08;
      =     "MAL1S033".Gr.All.Spare04;

//- Little help for PIC-People, Number 3
      UN    "G291M".Gr.InManual; // LIFTING DEVICE KILN 2
      UN    "G292M".Gr.InManual; // TRAVELLING DRIVE KILN 2
      UN    "G293M".Gr.InManual; // UNLOADING / LOADING SCREW KILN 2
      UN    "G294M".Gr.InManual; // DISCHARGE DOOR KILN 2
      UN    "G297M".Gr.InManual; // FAN KILN 2
      UN    "G298M".Gr.InManual; // FRESH AIR LOUVER KILN 2
      UN    "G299M".Gr.InManual; // RECYCLING AIR LOUVER KILN 2
      UN    "G300M".Gr.InManual; // EXHAUST AIR LOUVER KILN 2
      UN    "G302M".Gr.InManual; // HEATING KILN 2
      UN    "G303M".Gr.InManual; // LOUVER AIR HEATER 1 FOR KILN 2
      UN    "G304M".Gr.InManual; // WITHERING AIR KILN 2
      UN    "G279M".Gr.InManual; // HEATING KILN 1 + 2
      FP    DB923.DBX 2999.0;
      =     DB923.DBX 2999.1;
      U     DB923.DBX 2999.1;
      SPBN  RSM3;
      L     0;
      T     "MAL1S033Par".Ilo.Code_ILO_Funktion0; // FCM 32 LINE 1 SEC 32 KILN
      T     "MAL1S033Par".Ilo.ILOMode;
RSM3: NOP   0;

//- Combination OLD and NEW ---
      U     "MAL1S033".SecAc.Sta1On.Inf08;
      SPBN  IFM;
      L     "MAL1S033Par".Ilo.ILOMode;
      L     100;
      *I    ;
      T     "MAL1S033Par".Ilo.Code_ILO_Funktion0;
IFM:  NOP   0;

//  no ILO-mode >> cmd manual off to all used groups and reset all flags
      U     "MAL1S033".SecAc.Sta1On.Inf08;
      FN    "MAL1S033Par".Ilo.Flag.EdgeILOModeOn;
      S     "MAL1S033Par".Ilo.GrCMDManOff[1]; // (ManOff)
      R     "MAL1S033Par".Ilo.GrCMDManAdditional.Cmd1[1];
      R     "MAL1S033Par".Ilo.GrCMDManAdditional.Cmd2[2];
//  Gr-cmd manual OFF
      S     "G291M".Gr.CmdManualOff; // LIFTING DEVICE KILN 2
      S     "G292M".Gr.CmdManualOff; // TRAVELLING DRIVE KILN 2
      S     "G293M".Gr.CmdManualOff; // UNLOADING / LOADING SCREW KILN 2
      S     "G294M".Gr.CmdManualOff; // DISCHARGE DOOR KILN 2
      S     "G297M".Gr.CmdManualOff; // FAN KILN 2
      S     "G298M".Gr.CmdManualOff; // FRESH AIR LOUVER KILN 2
      S     "G299M".Gr.CmdManualOff; // RECYCLING AIR FLAP KILN 2
      S     "G302M".Gr.CmdManualOff; // HEATING KILN 2
      S     "G303M".Gr.CmdManualOff; // LOUVER AIR HEATER KILN 2
      S     "G304M".Gr.CmdManualOff; // WITHERING AIR KILN 2
      S     "G305M".Gr.CmdManualOff; // CHAIN CONVEYOR 9002 KILN 2
      S     "G279M".Gr.CmdManualOff; // HEATING KILN 1 + 2
//  RESET ADDITIONAL CMD`S
      R     "G291M".USW14; // ILO-cmd
      R     "G291M".USW15; // ILO-cmd
      R     "G292M".USW14; // ILO-cmd
      R     "G292M".USW15; // ILO-cmd
      R     "G293M".USW14; // ILO-cmd
      R     "G293M".USW15; // ILO-cmd
      R     "G294M".USW14; // ILO-cmd
      R     "G294M".USW15; // ILO-cmd
      R     "G297M".USW14; // ILO-cmd
      R     "G297M".USW15; // ILO-cmd
      R     "G298M".USW14; // ILO-cmd
      R     "G298M".USW15; // ILO-cmd
      R     "G299M".USW14; // ILO-cmd
      R     "G299M".USW15; // ILO-cmd
      R     "G302M".USW14; // ILO-cmd
      R     "G302M".USW15; // ILO-cmd
      R     "G303M".USW14; // ILO-cmd
      R     "G303M".USW15; // ILO-cmd
      R     "G304M".USW14; // ILO-cmd
      R     "G304M".USW15; // ILO-cmd
      R     "G305M".USW14; // ILO-cmd
      R     "G305M".USW15; // ILO-cmd
      R     "G279M".USW14; // ILO-cmd
      R     "G279M".USW15; // ILO-cmd

      NOP   0;
// --- FCM 01 - Lifting devices ---
      L     "MAL1S033Par".Ilo.ILOMode;
      L     1;
      <>I   ;
      SPB   IO1;
// man on
      U     "MAL1S033Par".Ilo.GrCMDManOn[1];
      S     "G291M".Gr.InManual; // LIFTING DEVICE KILN 2
      R     "MAL1S033Par".Ilo.GrCMDManOn[1];
// man off
      U     "MAL1S033Par".Ilo.GrCMDManOff[1];
      S     "G291M".Gr.CmdManualOff; // LIFTING DEVICE KILN 2
      R     "G291M".Gr.InManual; // LIFTING DEVICE KILN 2
      R     "G291M".USW14; // ILO-cmd
      R     "G291M".USW15; // ILO-cmd
      R     "MAL1S033Par".Ilo.GrCMDManOff[1];
      R     "MAL1S033Par".Ilo.GrCMDManAdditional.Cmd1[1];
      R     "MAL1S033Par".Ilo.GrCMDManAdditional.Cmd2[1];
// man start
      U     "MAL1S033Par".Ilo.GrCMDManStart[1];
      S     "G291M".Gr.CmdOn; // LIFTING DEVICE KILN 2
      S     "G291M".Gr.CmdContinue; // LIFTING DEVICE KILN 2
      R     "MAL1S033Par".Ilo.GrCMDManStart[1];
      U     "MAL1S033Par".Ilo.GrCMDManStart[2];
      R     "MAL1S033Par".Ilo.GrCMDManStart[2];
// man stop
      U     "MAL1S033Par".Ilo.GrCMDManStop[1];
      S     "G291M".Gr.CmdOff; // LIFTING DEVICE KILN 2
      R     "MAL1S033Par".Ilo.GrCMDManStop[1];
// man fault reset
      U     "MAL1S033Par".Ilo.GrCMDManFaultReset[1];
      S     "G291M".Gr.CmdFaultReset; // LIFTING DEVICE KILN 2
      R     "MAL1S033Par".Ilo.GrCMDManFaultReset[1];
// moving direction
      UN    "G291M".Gr.InManual; // LIFTING DEVICE KILN 2
      O(    ;
      L     "MAL1S033Par".Ilo.Code_ILO_Funktion0;
      L     100;
      <>I   ;
      )     ;
      SPB   Stat;
      UN    "MAL1S033Par".Ilo.GrCMDManAdditional.Cmd1[1];
      UN    "MAL1S033Par".Ilo.GrCMDManAdditional.Cmd2[1];
      L     "MAL1S033Par".Par.MachineValue.SOLLWERT_HUBZUG1_HOEHE;
      SPB   Tpos;
      U     "MAL1S033Par".Ilo.GrCMDManAdditional.Cmd1[1]; // ManUp
      L     2000; // 1850mm + Offset = 2000mm
      SPB   Tpos;
      U     "MAL1S033Par".Ilo.GrCMDManAdditional.Cmd2[1]; // ManDown
      L     0; // 0mm
      SPB   Tpos;
      SPA   Stat;
// target position
Tpos: NOP   0;
      T     "MAL1S033Par".Par.ParIntProcess.TarPos_ILO_LiftDev;
Stat: NOP   0;
IO1:  NOP   0;
      NOP   0;
// --- FCM 04 - Fans ---
      L     "MAL1S033Par".Ilo.ILOMode;
      L     4;
      <>I   ;
      SPB   IO4;
// man on
      U     "MAL1S033Par".Ilo.GrCMDManOn[1];
      S     "G297M".Gr.InManual; // FAN KILN 2
      R     "MAL1S033Par".Ilo.GrCMDManOn[1];
// man off
      U     "MAL1S033Par".Ilo.GrCMDManOff[1];
      S     "G297M".Gr.CmdManualOff; // FAN KILN 2
      R     "G297M".Gr.InManual; // FAN KILN 2
      R     "G297M".USW14; // ILO-cmd
      R     "G297M".USW15; // ILO-cmd
      R     "MAL1S033Par".Ilo.GrCMDManOff[1];
      R     "MAL1S033Par".Ilo.GrCMDManAdditional.Cmd1[1];
      R     "MAL1S033Par".Ilo.GrCMDManAdditional.Cmd2[1];
// man start
      U     "MAL1S033Par".Ilo.GrCMDManStart[1];
      S     "G297M".Gr.CmdOn; // FAN KILN 2
      S     "G297M".Gr.CmdContinue; // FAN KILN 2
      R     "MAL1S033Par".Ilo.GrCMDManStart[1];
      U     "MAL1S033Par".Ilo.GrCMDManStart[2];
      R     "MAL1S033Par".Ilo.GrCMDManStart[2];
// man stop
      U     "MAL1S033Par".Ilo.GrCMDManStop[1];
      S     "G297M".Gr.CmdOff; // FAN KILN 2
      R     "MAL1S033Par".Ilo.GrCMDManStop[1];
// man fault reset
      U     "MAL1S033Par".Ilo.GrCMDManFaultReset[1];
      S     "G297M".Gr.CmdFaultReset; // FAN KILN 2
      R     "MAL1S033Par".Ilo.GrCMDManFaultReset[1];
// target position
      UN    "G297M".Gr.InManual; // FAN KILN 2
      O(    ;
      L     "MAL1S033Par".Ilo.Code_ILO_Funktion0;
      L     400;
      <>I   ;
      )     ;
      SPB   F04a;
      L     "MAL1S033Par".Ilo.SetpointInt01[1];
      T     "MAL1S033Par".Par.ParIntProcess.Speed_ILO_Fan;
F04a: NOP   0;

IO4:  NOP   0;
      NOP   0;
// --- FCM 05 - Fans with target air temperature ---
      L     "MAL1S033Par".Ilo.ILOMode;
      L     5;
      <>I   ;
      SPB   IO5;
// man on
      U     "MAL1S033Par".Ilo.GrCMDManOn[1];
      S     "G297M".Gr.InManual; // FAN KILN 2
      S     "G299M".Gr.InManual; // RECYCLING AIR FLAP KILN 2
      S     "G299M".Gr.CmdOn; // No Button: RECYCLING AIR FLAP KILN 2
      S     "G299M".Gr.CmdContinue; // No Button RECYCLING AIR FLAP KILN 2
      S     "G302M".Gr.InManual; // HEATING KILN 2
      S     "G302M".Gr.CmdOn; // No Button: HEATING KILN 2
      S     "G302M".Gr.CmdContinue; // No Button HEATING KILN 2
      S     "G303M".Gr.InManual; // LOUVER AIR HEATER KILN 2
      S     "G303M".Gr.CmdOn; // No Button: LOUVER AIR HEATER KILN 2
      S     "G303M".Gr.CmdContinue; // No Button LOUVER AIR HEATER KILN 2
      S     "G298M".Gr.InManual; // FRESH AIR LOUVER KILN 2
      S     "G298M".Gr.CmdOn; // No Button: FRESH AIR LOUVER KILN 2
      S     "G298M".Gr.CmdContinue; // No Button FRESH AIR LOUVER KILN 2
      S     "G304M".Gr.InManual; // WITHERING AIR KILN 2
      S     "G304M".Gr.CmdOn; // No Button: WITHERING AIR KILN 2
      S     "G304M".Gr.CmdContinue; // No Button WITHERING AIR KILN 2
      R     "MAL1S033Par".Ilo.GrCMDManOn[1];
// man off
      U     "MAL1S033Par".Ilo.GrCMDManOff[1];
      S     "G297M".Gr.CmdManualOff; // FAN KILN 2
      R     "G297M".Gr.InManual; // FAN KILN 2
      R     "G297M".USW14; // ILO-cmd
      R     "G297M".USW15; // ILO-cmd
      S     "G299M".Gr.CmdManualOff; // RECYCLING AIR FLAP KILN 2
      R     "G299M".Gr.InManual; // RECYCLING AIR FLAP KILN 2
      R     "G299M".USW14; // ILO-cmd
      R     "G299M".USW15; // ILO-cmd
      S     "G302M".Gr.CmdManualOff; // HEATING KILN 2
      R     "G302M".Gr.InManual; // HEATING KILN 2
      R     "G302M".USW14; // ILO-cmd
      R     "G302M".USW15; // ILO-cmd
      S     "G303M".Gr.CmdManualOff; // LOUVER AIR HEATER KILN 2
      R     "G303M".Gr.InManual; // LOUVER AIR HEATER KILN 2
      R     "G303M".USW14; // ILO-cmd
      R     "G303M".USW15; // ILO-cmd
      S     "G298M".Gr.CmdManualOff; // FRESH AIR LOUVER KILN 2
      R     "G298M".Gr.InManual; // FRESH AIR LOUVER KILN 2
      R     "G298M".USW14; // ILO-cmd
      R     "G298M".USW15; // ILO-cmd
      S     "G304M".Gr.CmdManualOff; // WITHERING AIR KILN 2
      R     "G304M".Gr.InManual; // WITHERING AIR KILN 2
      R     "G304M".USW14; // ILO-cmd
      R     "G304M".USW15; // ILO-cmd
      R     "MAL1S033Par".Ilo.GrCMDManOff[1];
      R     "MAL1S033Par".Ilo.GrCMDManAdditional.Cmd1[1];
      R     "MAL1S033Par".Ilo.GrCMDManAdditional.Cmd2[1];
// man start
      U     "MAL1S033Par".Ilo.GrCMDManStart[1];
      S     "G297M".Gr.CmdOn; // FAN KILN 2
      S     "G297M".Gr.CmdContinue; // FAN KILN 2
      S     "G299M".Gr.CmdOn; // RECYCLING AIR FLAP KILN 2
      S     "G299M".Gr.CmdContinue; // RECYCLING AIR FLAP KILN 2
      S     "G302M".Gr.CmdOn; // HEATING KILN 2
      S     "G302M".Gr.CmdContinue; // HEATING KILN 2
      S     "G303M".Gr.CmdOn; // LOUVER AIR HEATER KILN 2
      S     "G303M".Gr.CmdContinue; // LOUVER AIR HEATER KILN 2
      S     "G298M".Gr.CmdOn; // FRESH AIR LOUVER KILN 2
      S     "G298M".Gr.CmdContinue; // FRESH AIR LOUVER KILN 2
      S     "G304M".Gr.CmdOn; // WITHERING AIR KILN 2
      S     "G304M".Gr.CmdContinue; // WITHERING AIR KILN 2
      R     "MAL1S033Par".Ilo.GrCMDManStart[1];
      U     "MAL1S033Par".Ilo.GrCMDManStart[2];
      R     "MAL1S033Par".Ilo.GrCMDManStart[2];
// man stop
      U     "MAL1S033Par".Ilo.GrSTMan[17];
      S     "G297M".Gr.CmdOff; // FAN KILN 2
      S     "G299M".Gr.CmdOff; // RECYCLING AIR FLAP KILN 2
      S     "G302M".Gr.CmdOff; // HEATING KILN 2
      S     "G303M".Gr.CmdOff; // LOUVER AIR HEATER KILN 2
      S     "G298M".Gr.CmdOff; // FRESH AIR LOUVER KILN 2
      S     "G304M".Gr.CmdOff; // WITHERING AIR KILN 2
      R     "MAL1S033Par".Ilo.GrSTMan[17];
// man fault reset
      U     "MAL1S033Par".Ilo.GrCMDManFaultReset[1];
      S     "G297M".Gr.CmdFaultReset; // FAN KILN 2
      S     "G299M".Gr.CmdFaultReset; // RECYCLING AIR FLAP KILN 2
      S     "G302M".Gr.CmdFaultReset; // HEATING KILN 2
      S     "G303M".Gr.CmdFaultReset; // LOUVER AIR HEATER KILN 2
      S     "G298M".Gr.CmdFaultReset; // FRESH AIR LOUVER KILN 2
      S     "G304M".Gr.CmdFaultReset; // WITHERING AIR KILN 2
      R     "MAL1S033Par".Ilo.GrCMDManFaultReset[1];
// target position
      UN    "G297M".Gr.InManual; // FAN KILN 2
      O(    ;
      L     "MAL1S033Par".Ilo.Code_ILO_Funktion0;
      L     500;
      <>I   ;
      )     ;
      SPB   F05b;
      L     "MAL1S033Par".Ilo.SetpointInt01[1];
      T     "MAL1S033Par".Par.ParIntProcess.Speed_ILO_Fan;
F05b: NOP   0;
      UN    "G299M".Gr.InManual; // Recycling Air Flap Kilningbox 1
      O(    ;
      L     "MAL1S033Par".Ilo.Code_ILO_Funktion0;
      L     500;
      <>I   ;
      )     ;
      SPB   F05c;
      L     "MAL1S033Par".Ilo.SetpointInt03[1];
      T     "MAL1S033Par".Par.ParIntProcess.TarPos_ILO_RecycAir;
F05c: NOP   0;
      UN    "G304M".Gr.InManual; // Withering Air Flap Kilningbox 1
      O(    ;
      L     "MAL1S033Par".Ilo.Code_ILO_Funktion0;
      L     500;
      <>I   ;
      )     ;
      SPB   F05d;
      L     "MAL1S033Par".Ilo.SetpointInt04[1];
      T     "MAL1S033Par".Par.ParIntProcess.TarPos_ILO_WitheringAir;
F05d: NOP   0;
      UN    "G302M".Gr.InManual; // Heating Kiln 2
      O(    ;
      L     "MAL1S033Par".Ilo.Code_ILO_Funktion0;
      L     500;
      <>I   ;
      )     ;
      SPB   F05e;
      L     "MAL1S033Par".Ilo.SetpointInt01[2];
      T     "MAL1S033Par".Par.ParIntProcess.TargetTemperature_ILO;
F05e: NOP   0;

IO5:  NOP   0;
      NOP   0;
// --- FCM 06 - Fresh air flap ---
      L     "MAL1S033Par".Ilo.ILOMode;
      L     6;
      <>I   ;
      SPB   IO6;
// man on
      U     "MAL1S033Par".Ilo.GrCMDManOn[1];
      S     "G298M".Gr.InManual; // FRESH AIR LOUVER KILN 2
      R     "MAL1S033Par".Ilo.GrCMDManOn[1];
// man off
      U     "MAL1S033Par".Ilo.GrCMDManOff[1];
      S     "G298M".Gr.CmdManualOff; // FRESH AIR LOUVER KILN 2
      R     "G298M".Gr.InManual; // FRESH AIR LOUVER KILN 2
      R     "G298M".USW14; // ILO-cmd
      R     "G298M".USW15; // ILO-cmd
      R     "MAL1S033Par".Ilo.GrCMDManOff[1];
      R     "MAL1S033Par".Ilo.GrCMDManAdditional.Cmd1[1];
      R     "MAL1S033Par".Ilo.GrCMDManAdditional.Cmd2[1];
// man start
      U     "MAL1S033Par".Ilo.GrCMDManStart[1];
      S     "G298M".Gr.CmdOn; // FRESH AIR LOUVER KILN 2
      S     "G298M".Gr.CmdContinue; // FRESH AIR LOUVER KILN 2
      R     "MAL1S033Par".Ilo.GrCMDManStart[1];
      U     "MAL1S033Par".Ilo.GrCMDManStart[2];
      R     "MAL1S033Par".Ilo.GrCMDManStart[2];
// man stop
      U     "MAL1S033Par".Ilo.GrCMDManStop[1];
      S     "G298M".Gr.CmdOff; // FRESH AIR LOUVER KILN 2
      R     "MAL1S033Par".Ilo.GrCMDManStop[1];
// man fault reset
      U     "MAL1S033Par".Ilo.GrCMDManFaultReset[1];
      S     "G298M".Gr.CmdFaultReset; // FRESH AIR LOUVER KILN 2
      R     "MAL1S033Par".Ilo.GrCMDManFaultReset[1];
// moving direction

// target position
      UN    "G298M".Gr.InManual; // FRESH AIR LOUVER KILN 2
      SPB   F06b;
      L     "MAL1S033Par".Ilo.SetpointInt01[1];
      T     "MAL1S033Par".Par.ParIntProcess.TarPos_ILO_FreshAir;
F06b: NOP   0;

IO6:  NOP   0;
      NOP   0;
// --- FCM 07 - Recycling air flap ---
      L     "MAL1S033Par".Ilo.ILOMode;
      L     7;
      <>I   ;
      SPB   IO7;
// man on
      U     "MAL1S033Par".Ilo.GrCMDManOn[1];
      S     "G299M".Gr.InManual; // RECYCLING AIR FLAP KILN 2
      S     "G304M".Gr.InManual; // WITHERING AIR KILN 2
      R     "MAL1S033Par".Ilo.GrCMDManOn[1];
// man off
      U     "MAL1S033Par".Ilo.GrCMDManOff[1];
      S     "G299M".Gr.CmdManualOff; // RECYCLING AIR FLAP KILN 2
      R     "G299M".Gr.InManual; // RECYCLING AIR FLAP KILN 2
      R     "G299M".USW14; // ILO-cmd
      R     "G299M".USW15; // ILO-cmd
      S     "G304M".Gr.CmdManualOff; // WITHERING AIR KILN 2
      R     "G304M".Gr.InManual; // WITHERING AIR KILN 2
      R     "G304M".USW14; // ILO-cmd
      R     "G304M".USW15; // ILO-cmd
      R     "MAL1S033Par".Ilo.GrCMDManOff[1];
      R     "MAL1S033Par".Ilo.GrCMDManAdditional.Cmd1[1];
      R     "MAL1S033Par".Ilo.GrCMDManAdditional.Cmd2[1];
// man start
      U     "MAL1S033Par".Ilo.GrCMDManStart[1];
      S     "G299M".Gr.CmdOn; // RECYCLING AIR FLAP KILN 2
      S     "G299M".Gr.CmdContinue; // RECYCLING AIR FLAP KILN 2
      S     "G304M".Gr.CmdOn; // WITHERING AIR KILN 2
      S     "G304M".Gr.CmdContinue; // WITHERING AIR KILN 2
      R     "MAL1S033Par".Ilo.GrCMDManStart[1];
      U     "MAL1S033Par".Ilo.GrCMDManStart[2];
      R     "MAL1S033Par".Ilo.GrCMDManStart[2];
// man stop
      U     "MAL1S033Par".Ilo.GrCMDManStop[1];
      S     "G299M".Gr.CmdOff; // RECYCLING AIR FLAP KILN 2
      S     "G304M".Gr.CmdOff; // WITHERING AIR KILN 2
      R     "MAL1S033Par".Ilo.GrCMDManStop[1];
// man fault reset
      U     "MAL1S033Par".Ilo.GrCMDManFaultReset[1];
      S     "G299M".Gr.CmdFaultReset; // RECYCLING AIR FLAP KILN 2
      S     "G304M".Gr.CmdFaultReset; // WITHERING AIR KILN 2
      R     "MAL1S033Par".Ilo.GrCMDManFaultReset[1];
// moving direction

// target position
      UN    "G299M".Gr.InManual; // RECYCLING AIR FLAP KILN 2
      SPB   F07a;
      L     "MAL1S033Par".Ilo.SetpointInt01[1];
      T     "MAL1S033Par".Par.ParIntProcess.TarPos_ILO_RecycAir;
F07a: NOP   0;
IO7:  NOP   0;
      NOP   0;
// --- FCM 09 - Floor drives ---
      L     "MAL1S033Par".Ilo.ILOMode;
      L     9;
      <>I   ;
      SPB   IO9;
// man on
      U     "MAL1S033Par".Ilo.GrCMDManOn[1];
      S     "G292M".Gr.InManual; // TRAVELLING DRIVE KILN 2
      R     "MAL1S033Par".Ilo.GrCMDManOn[1];
// man off
      U     "MAL1S033Par".Ilo.GrCMDManOff[1];
      S     "G292M".Gr.CmdManualOff; // TRAVELLING DRIVE KILN 2
      R     "G292M".Gr.InManual; // TRAVELLING DRIVE KILN 2
      R     "G292M".USW14; // ILO-cmd
      R     "G292M".USW15; // ILO-cmd
      R     "MAL1S033Par".Ilo.GrCMDManOff[1];
      R     "MAL1S033Par".Ilo.GrCMDManAdditional.Cmd1[1];
      R     "MAL1S033Par".Ilo.GrCMDManAdditional.Cmd2[1];
// man start
      U     "MAL1S033Par".Ilo.GrCMDManStart[1];
      S     "G292M".Gr.CmdOn; // TRAVELLING DRIVE KILN 2
      S     "G292M".Gr.CmdContinue; // TRAVELLING DRIVE KILN 2
      R     "MAL1S033Par".Ilo.GrCMDManStart[1];
      U     "MAL1S033Par".Ilo.GrCMDManStart[2];
      R     "MAL1S033Par".Ilo.GrCMDManStart[2];
// man stop
      U     "MAL1S033Par".Ilo.GrCMDManStop[1];
      S     "G292M".Gr.CmdOff; // TRAVELLING DRIVE KILN 2
      R     "MAL1S033Par".Ilo.GrCMDManStop[1];
// man fault reset
      U     "MAL1S033Par".Ilo.GrCMDManOn[17];
      S     "G292M".Gr.CmdFaultReset; // TRAVELLING DRIVE KILN 2
      R     "MAL1S033Par".Ilo.GrCMDManOn[17];
      NOP   0;
      UN    "G292M".Gr.InManual; // TRAVELLING DRIVE KILN 2
      O     ;
      UN    "MAL1S033Par".Ilo.GrCMDManAdditional.Cmd1[1];
      UN    "MAL1S033Par".Ilo.GrCMDManAdditional.Cmd2[1];
      SPB   f092;
      U     "MAL1S033Par".Ilo.GrCMDManAdditional.Cmd1[1];
      =     "G292M".USW14; // ILO-cmd run fwd
      U     "MAL1S033Par".Ilo.GrCMDManAdditional.Cmd2[1];
      =     "G292M".USW15; // ILO-cmd run rev
// target position
      L     "MAL1S033Par".Ilo.SetpointInt01[1];
      T     "MAL1S033Par".Par.ParIntProcess.Speed_ILO_FloorRotating;
f092: NOP   0;

IO9:  NOP   0;
      NOP   0;
// --- FCM 10 - Floor drives and lifting devices ---
      L     "MAL1S033Par".Ilo.ILOMode;
      L     10;
      <>I   ;
      SPB   IO10;
// man on
      U     "MAL1S033Par".Ilo.GrCMDManOn[1];
      S     "G291M".Gr.InManual; // LIFTING DEVICE KILN 2
      S     "G291M".Gr.CmdOn; // No Button: LIFTING DEVICE KILN 2
      S     "G291M".Gr.CmdContinue; // No Button LIFTING DEVICE KILN 2
      S     "G292M".Gr.InManual; // TRAVELLING DRIVE KILN 2
      R     "MAL1S033Par".Ilo.GrCMDManOn[1];
// man off
      U     "MAL1S033Par".Ilo.GrCMDManOff[1];
      S     "G291M".Gr.CmdManualOff; // LIFTING DEVICE KILN 2
      R     "G291M".Gr.InManual; // LIFTING DEVICE KILN 2
      R     "G291M".USW14; // ILO-cmd
      R     "G291M".USW15; // ILO-cmd
      S     "G292M".Gr.CmdManualOff; // TRAVELLING DRIVE KILN 2
      R     "G292M".Gr.InManual; // TRAVELLING DRIVE KILN 2
      R     "G292M".USW14; // ILO-cmd
      R     "G292M".USW15; // ILO-cmd
      R     "MAL1S033Par".Ilo.GrCMDManOff[1];
      R     "MAL1S033Par".Ilo.GrCMDManAdditional.Cmd1[1];
      R     "MAL1S033Par".Ilo.GrCMDManAdditional.Cmd2[1];
// man start
      U     "MAL1S033Par".Ilo.GrCMDManStart[1];
      S     "G292M".Gr.CmdOn; // TRAVELLING DRIVE KILN 2
      S     "G292M".Gr.CmdContinue; // TRAVELLING DRIVE KILN 2
      R     "MAL1S033Par".Ilo.GrCMDManStart[1];
      U     "MAL1S033Par".Ilo.GrCMDManStart[2];
      S     "G291M".Gr.CmdOn; // LIFTING DEVICE KILN 2
      S     "G291M".Gr.CmdContinue; // LIFTING DEVICE KILN 2
      R     "MAL1S033Par".Ilo.GrCMDManStart[2];
      U     "MAL1S033Par".Ilo.GrCMDManStart[3];
      R     "MAL1S033Par".Ilo.GrCMDManStart[3];
// man stop
      U     "MAL1S033Par".Ilo.GrCMDManStop[1];
      S     "G291M".Gr.CmdOff; // LIFTING DEVICE KILN 2
      S     "G292M".Gr.CmdOff; // TRAVELLING DRIVE KILN 2
      R     "MAL1S033Par".Ilo.GrCMDManStop[1];
// man fault reset
      U     "MAL1S033Par".Ilo.GrCMDManFaultReset[1];
      S     "G291M".Gr.CmdFaultReset; // LIFTING DEVICE KILN 2
      S     "G292M".Gr.CmdFaultReset; // TRAVELLING DRIVE KILN 2
      R     "MAL1S033Par".Ilo.GrCMDManFaultReset[1];
// moving direction
      NOP   0;
      UN    "G292M".Gr.InManual; // TRAVELLING DRIVE KILN 2
      O     ;
      UN    "MAL1S033Par".Ilo.GrCMDManAdditional.Cmd1[1];
      UN    "MAL1S033Par".Ilo.GrCMDManAdditional.Cmd2[1];
      SPB   f102;
      U     "MAL1S033Par".Ilo.GrCMDManAdditional.Cmd1[1];
      =     "G292M".USW14; // ILO-cmd run fwd
      U     "MAL1S033Par".Ilo.GrCMDManAdditional.Cmd2[1];
      =     "G292M".USW15; // ILO-cmd run rev
// target speed floor drives
      L     "MAL1S033Par".Ilo.SetpointInt01[1];
      T     "MAL1S033Par".Par.ParIntProcess.Speed_ILO_FloorRotating;
f102: NOP   0;
      UN    "G291M".Gr.InManual; // LIFTING DEVICE KILN 2
      O(    ;
      L     "MAL1S033Par".Ilo.Code_ILO_Funktion0;
      L     1000;
      <>I   ;
      )     ;
      SPB   f103;
// target position lifting devices
      L     "MAL1S033Par".Ilo.SetpointInt02[1];
      T     "MAL1S033Par".Par.ParIntProcess.TarPos_ILO_LiftDev;
f103: NOP   0;

IO10: NOP   0;
      NOP   0;
// --- FCM 11 - Floor drives and lifting devices and screw ---
      L     "MAL1S033Par".Ilo.ILOMode;
      L     11;
      <>I   ;
      SPB   IO11;
// man on
      U     "MAL1S033Par".Ilo.GrCMDManOn[1];
      S     "G291M".Gr.InManual; // LIFTING DEVICE KILN 2
      S     "G291M".Gr.CmdOn; // No Button: LIFTING DEVICE KILN 2
      S     "G291M".Gr.CmdContinue; // No Button LIFTING DEVICE KILN 2
      S     "G292M".Gr.InManual; // TRAVELLING DRIVE KILN 2
      S     "G293M".Gr.InManual; // UNLOADING / LOADING SCREW KILN 2
      R     "MAL1S033Par".Ilo.GrCMDManOn[1];
// man off
      U     "MAL1S033Par".Ilo.GrCMDManOff[1];
      S     "G291M".Gr.CmdManualOff; // LIFTING DEVICE KILN 2
      R     "G291M".Gr.InManual; // LIFTING DEVICE KILN 2
      R     "G291M".USW14; // ILO-cmd
      R     "G291M".USW15; // ILO-cmd
      S     "G292M".Gr.CmdManualOff; // TRAVELLING DRIVE KILN 2
      R     "G292M".Gr.InManual; // TRAVELLING DRIVE KILN 2
      R     "G292M".USW14; // ILO-cmd
      R     "G292M".USW15; // ILO-cmd
      S     "G293M".Gr.CmdManualOff; // UNLOADING / LOADING SCREW KILN 2
      R     "G293M".Gr.InManual; // UNLOADING / LOADING SCREW KILN 2
      R     "G293M".USW14; // ILO-cmd
      R     "G293M".USW15; // ILO-cmd
      R     "MAL1S033Par".Ilo.GrCMDManOff[1];
      R     "MAL1S033Par".Ilo.GrCMDManAdditional.Cmd1[1];
      R     "MAL1S033Par".Ilo.GrCMDManAdditional.Cmd2[1];
// man start
      U     "MAL1S033Par".Ilo.GrCMDManStart[1];
      S     "G292M".Gr.CmdOn; // TRAVELLING DRIVE KILN 2
      S     "G292M".Gr.CmdContinue; // TRAVELLING DRIVE KILN 2
      R     "MAL1S033Par".Ilo.GrCMDManStart[1];
      U     "MAL1S033Par".Ilo.GrCMDManStart[2];
      S     "G291M".Gr.CmdOn; // LIFTING DEVICE KILN 2
      S     "G291M".Gr.CmdContinue; // LIFTING DEVICE KILN 2
      R     "MAL1S033Par".Ilo.GrCMDManStart[2];
      U     "MAL1S033Par".Ilo.GrCMDManStart[3];
      S     "G293M".Gr.CmdOn; // UNLOADING / LOADING SCREW KILN 2
      S     "G293M".Gr.CmdContinue; // UNLOADING / LOADING SCREW KILN 2
      R     "MAL1S033Par".Ilo.GrCMDManStart[3];
      U     "MAL1S033Par".Ilo.GrCMDManStart[4];
      S     "G293M".Gr.CmdOn; // UNLOADING / LOADING SCREW KILN 2
      S     "G293M".Gr.CmdContinue; // UNLOADING / LOADING SCREW KILN 2
      R     "MAL1S033Par".Ilo.GrCMDManStart[4];
// man stop
      U     "MAL1S033Par".Ilo.GrCMDManStop[1];
      S     "G291M".Gr.CmdOff; // LIFTING DEVICE KILN 2
      S     "G292M".Gr.CmdOff; // TRAVELLING DRIVE KILN 2
      S     "G293M".Gr.CmdOff; // UNLOADING / LOADING SCREW KILN 2
      R     "MAL1S033Par".Ilo.GrCMDManStop[1];
// man fault reset
      U     "MAL1S033Par".Ilo.GrCMDManFaultReset[1];
      S     "G291M".Gr.CmdFaultReset; // LIFTING DEVICE KILN 2
      S     "G292M".Gr.CmdFaultReset; // TRAVELLING DRIVE KILN 2
      S     "G293M".Gr.CmdFaultReset; // UNLOADING / LOADING SCREW KILN 2
      R     "MAL1S033Par".Ilo.GrCMDManFaultReset[1];
// moving direction
      UN    "G292M".Gr.InManual; // TRAVELLING DRIVE KILN 2
      O     ;
      UN    "MAL1S033Par".Ilo.GrCMDManAdditional.Cmd1[1];
      UN    "MAL1S033Par".Ilo.GrCMDManAdditional.Cmd2[1];
      SPB   f112;
      U     "MAL1S033Par".Ilo.GrCMDManAdditional.Cmd1[1];
      =     "G292M".USW14; // ILO-cmd run fwd
      U     "MAL1S033Par".Ilo.GrCMDManAdditional.Cmd2[1];
      =     "G292M".USW15; // ILO-cmd run rev
// target speed floor drives
      L     "MAL1S033Par".Ilo.SetpointInt01[1];
      T     "MAL1S033Par".Par.ParIntProcess.Speed_ILO_FloorRotating;
f112: NOP   0;
      UN    "G291M".Gr.InManual; // Malting Plant OAO Belsolod Ivanonvo Weissrussland
      O(    ;
      L     "MAL1S033Par".Ilo.Code_ILO_Funktion0;
      L     1100;
      <>I   ;
      )     ;
      SPB   f113;
// target position lifting devices
      L     "MAL1S033Par".Ilo.SetpointInt01[2];
      L     "MAL1S033Par".Ilo.SetpointInt02[1];
      T     "MAL1S033Par".Par.ParIntProcess.TarPos_ILO_LiftDev;
f113: NOP   0;
      UN    "G293M".Gr.InManual; // UNLOADING / LOADING SCREW KILN 2
      O     ;
      UN    "MAL1S033Par".Ilo.GrCMDManAdditional.Cmd1[3];
      UN    "MAL1S033Par".Ilo.GrCMDManAdditional.Cmd2[3];
      SPB   f114;
      U     "MAL1S033Par".Ilo.GrCMDManAdditional.Cmd1[3];
      =     "G293M".USW14; // ILO-cmd run fwd
      U     "MAL1S033Par".Ilo.GrCMDManAdditional.Cmd2[3];
      =     "G293M".USW15; // ILO-cmd run rev
f114: NOP   0;
IO11: NOP   0;
      NOP   0;
// --- FCM 12 - Floor drives and lifting devices and screw and discharging flap ---
      L     "MAL1S033Par".Ilo.ILOMode;
      L     12;
      <>I   ;
      SPB   IO12;
// man on
      U     "MAL1S033Par".Ilo.GrCMDManOn[1];
      S     "G291M".Gr.InManual; // LIFTING DEVICE KILN 2
      S     "G291M".Gr.CmdOn; // No Button: LIFTING DEVICE KILN 2
      S     "G291M".Gr.CmdContinue; // No Button LIFTING DEVICE KILN 2
      S     "G292M".Gr.InManual; // TRAVELLING DRIVE KILN 2
      S     "G293M".Gr.InManual; // UNLOADING / LOADING SCREW KILN 2
      S     "G294M".Gr.InManual; // DISCHARGE DOOR KILN 2
      R     "MAL1S033Par".Ilo.GrCMDManOn[1];
// man off
      U     "MAL1S033Par".Ilo.GrCMDManOff[1];
      S     "G291M".Gr.CmdManualOff; // LIFTING DEVICE KILN 2
      R     "G291M".Gr.InManual; // LIFTING DEVICE KILN 2
      R     "G291M".USW14; // ILO-cmd
      R     "G291M".USW15; // ILO-cmd
      S     "G292M".Gr.CmdManualOff; // TRAVELLING DRIVE KILN 2
      R     "G292M".Gr.InManual; // TRAVELLING DRIVE KILN 2
      R     "G292M".USW14; // ILO-cmd
      R     "G292M".USW15; // ILO-cmd
      S     "G293M".Gr.CmdManualOff; // UNLOADING / LOADING SCREW KILN 2
      R     "G293M".Gr.InManual; // UNLOADING / LOADING SCREW KILN 2
      R     "G293M".USW14; // ILO-cmd
      R     "G293M".USW15; // ILO-cmd
      S     "G294M".Gr.CmdManualOff; // DISCHARGE DOOR KILN 2
      R     "G294M".Gr.InManual; // DISCHARGE DOOR KILN 2
      R     "G294M".USW14; // ILO-cmd
      R     "G294M".USW15; // ILO-cmd
      R     "MAL1S033Par".Ilo.GrCMDManOff[1];
      R     "MAL1S033Par".Ilo.GrCMDManAdditional.Cmd1[1];
      R     "MAL1S033Par".Ilo.GrCMDManAdditional.Cmd2[1];
// man start
      U     "MAL1S033Par".Ilo.GrCMDManStart[1];
      S     "G292M".Gr.CmdOn; // TRAVELLING DRIVE KILN 2
      S     "G292M".Gr.CmdContinue; // TRAVELLING DRIVE KILN 2
      R     "MAL1S033Par".Ilo.GrCMDManStart[1];
      U     "MAL1S033Par".Ilo.GrCMDManStart[2];
      S     "G291M".Gr.CmdOn; // LIFTING DEVICE KILN 2
      S     "G291M".Gr.CmdContinue; // LIFTING DEVICE KILN 2
      R     "MAL1S033Par".Ilo.GrCMDManStart[2];
      U     "MAL1S033Par".Ilo.GrCMDManStart[3];
      S     "G293M".Gr.CmdOn; // UNLOADING / LOADING SCREW KILN 2
      S     "G293M".Gr.CmdContinue; // UNLOADING / LOADING SCREW KILN 2
      R     "MAL1S033Par".Ilo.GrCMDManStart[3];
      U     "MAL1S033Par".Ilo.GrCMDManStart[4];
      S     "G293M".Gr.CmdOn; // UNLOADING / LOADING SCREW KILN 2
      S     "G293M".Gr.CmdContinue; // UNLOADING / LOADING SCREW KILN 2
      R     "MAL1S033Par".Ilo.GrCMDManStart[4];
// man stop
      U     "MAL1S033Par".Ilo.GrCMDManStop[1];
      S     "G291M".Gr.CmdOff; // LIFTING DEVICE KILN 2
      S     "G292M".Gr.CmdOff; // TRAVELLING DRIVE KILN 2
      S     "G293M".Gr.CmdOff; // UNLOADING / LOADING SCREW KILN 2
      S     "G294M".Gr.CmdOff; // DISCHARGE DOOR KILN 2
      R     "MAL1S033Par".Ilo.GrCMDManStop[1];
// man fault reset
      U     "MAL1S033Par".Ilo.GrCMDManFaultReset[1];
      S     "G291M".Gr.CmdFaultReset; // LIFTING DEVICE KILN 2
      S     "G292M".Gr.CmdFaultReset; // TRAVELLING DRIVE KILN 2
      S     "G293M".Gr.CmdFaultReset; // UNLOADING / LOADING SCREW KILN 2
      S     "G294M".Gr.CmdFaultReset; // DISCHARGE DOOR KILN 2
      R     "MAL1S033Par".Ilo.GrCMDManFaultReset[1];
// moving direction
      UN    "G292M".Gr.InManual; // TRAVELLING DRIVE KILN 2
      O     ;
      UN    "MAL1S033Par".Ilo.GrCMDManAdditional.Cmd1[1];
      UN    "MAL1S033Par".Ilo.GrCMDManAdditional.Cmd2[1];
      SPB   f122;
      U     "MAL1S033Par".Ilo.GrCMDManAdditional.Cmd1[1];
      =     "G292M".USW14; // ILO-cmd run fwd
      U     "MAL1S033Par".Ilo.GrCMDManAdditional.Cmd2[1];
      =     "G292M".USW15; // ILO-cmd run rev
// target speed floor drives
      L     "MAL1S033Par".Ilo.SetpointInt01[1];
      T     "MAL1S033Par".Par.ParIntProcess.Speed_ILO_FloorRotating;
f122: NOP   0;
      UN    "G291M".Gr.InManual; // LIFTING DEVICE KILN 2
      O(    ;
      L     "MAL1S033Par".Ilo.Code_ILO_Funktion0;
      L     1200;
      <>I   ;
      )     ;
      SPB   f123;
// target position lifting devices
      L     "MAL1S033Par".Ilo.SetpointInt01[18];
      T     "MAL1S033Par".Par.ParIntProcess.TarPos_ILO_LiftDev;
f123: NOP   0;
      UN    "G293M".Gr.InManual; // Malting Plant OAO Belsolod Ivanonvo Weissrussland
      O     ;
      UN    "MAL1S033Par".Ilo.GrCMDManAdditional.Cmd1[3];
      UN    "MAL1S033Par".Ilo.GrCMDManAdditional.Cmd2[3];
      SPB   f124;
      U     "MAL1S033Par".Ilo.GrCMDManAdditional.Cmd1[3];
      =     "G293M".USW14; // ILO-cmd run fwd
      U     "MAL1S033Par".Ilo.GrCMDManAdditional.Cmd2[3];
      =     "G293M".USW15; // ILO-cmd run rev
f124: NOP   0;
      UN    "G294M".Gr.InManual; // DISCHARGE DOOR KILN 2
      O     ;
      UN    "MAL1S033Par".Ilo.GrCMDManAdditional.Cmd1[4];
      UN    "MAL1S033Par".Ilo.GrCMDManAdditional.Cmd2[4];
      SPB   f125;
      U     "MAL1S033Par".Ilo.GrCMDManAdditional.Cmd1[4];
      =     "G294M".USW14; // ILO-cmd OPEN
      U     "MAL1S033Par".Ilo.GrCMDManAdditional.Cmd2[4];
      =     "G294M".USW15; // ILO-cmd CLOSE
f125: NOP   0;
IO12: NOP   0;
//
// copy state
      U     "G291M".Gr.InOutAutostartMan; // LIFTING DEVICE KILN 2
      =     "MAL1S033Par".Ilo.GrSTMan[1];
      U     "G292M".Gr.InOutAutostartMan; // TRAVELLING DRIVE KILN 2
      =     "MAL1S033Par".Ilo.GrSTMan[2];
      U     "G293M".Gr.InOutAutostartMan; // UNLOADING / LOADING SCREW KILN 2
      =     "MAL1S033Par".Ilo.GrSTMan[3];
      U     "G294M".Gr.InOutAutostartMan; // DISCHARGE DOOR KILN 2
      =     "MAL1S033Par".Ilo.GrSTMan[4];
      U     "G297M".Gr.InOutAutostartMan; // FAN KILN 2
      =     "MAL1S033Par".Ilo.GrSTMan[6];
      U     "G302M".Gr.InOutAutostartMan; // HEATING KILN 2
      =     "MAL1S033Par".Ilo.GrSTMan[11];
      U     "G303M".Gr.InOutAutostartMan; // LOUVER AIR HEATER KILN 2
      =     "MAL1S033Par".Ilo.GrSTMan[12];
      U     "G298M".Gr.InOutAutostartMan; // FRESH AIR LOUVER KILN 2
      =     "MAL1S033Par".Ilo.GrSTMan[13];
      U     "G304M".Gr.InOutAutostartMan; // WITHERING AIR KILN 2
      =     "MAL1S033Par".Ilo.GrSTMan[14];
      U     "G299M".Gr.InOutAutostartMan; // RECYCLING AIR FLAP KILN 2
      =     "MAL1S033Par".Ilo.GrSTMan[15];
      U     "G279M".Gr.InOutAutostartMan; // HEATING KILN 1 + 2
      =     "MAL1S033Par".Ilo.GrSTMan[16];
NETWORK
TITLE =ASW_9999: Init Flag
// clear all flags explicde to find them back
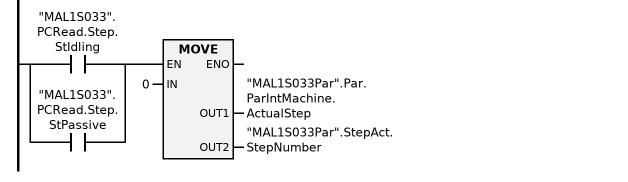
      U     "MAL1S033".PCRead.Step.StIdling;
      O     "MAL1S033".PCRead.Step.StPassive;
      R     "MAL1S033Par".Par.FlagFunction_1.StepLoading;
      R     "MAL1S033Par".Par.FlagFunction_1.StepUnloading;
      R     "MAL1S033Par".Par.FlagFunction_1.StepCleaning;
      R     "MAL1S033Par".Par.FlagFunction_1.LoadingBreak;
      R     "MAL1S033Par".Par.FlagFunction_1.UnloadingBreak;
      R     "MAL1S033Par".Par.FlagFunction_1.CleaningBreak;
      R     "MAL1S033Par".Par.FlagFunction_1.FinishLoading;
      R     "MAL1S033Par".Par.FlagFunction_1.FinishUnloading;
      R     "MAL1S033Par".Par.FlagFunction_1.FinishCleaning;
      R     "MAL1S033Par".Par.FlagFunction_1.Entladerunden_erreicht;
      R     "MAL1S033Par".Par.FlagFunction_1.Reinigungsrunde_erreicht;
      R     "MAL1S033Par".Par.FlagFunction_1.UnloadEnd;
      R     "MAL1S033Par".Par.FlagFunction_1.LoadEnd;
      R     "MAL1S033Par".Par.FlagFunction_1.UnloadFirstPart;
      R     "MAL1S033Par".Par.FlagFunction_1.UnloadSecondPart;
      R     "MAL1S033Par".Par.FlagProcess.ProcessActive;
      R     "MAL1S033Par".Par.FlagProcess.StartProzess_FP;
      R     "MAL1S033Par".Par.FlagProcess.StartProzess_SCAN;
      R     "MAL1S033Par".Par.FlagProcess.TurningFloor;
      R     "MAL1S033Par".Par.FlagProcess.Cooling_Activ;
      R     "MAL1S033Par".Par.FlagProcess.FP_SendResultToPIC;
      R     "MAL1S033Par".Par.FlagProcess.ProcessEnd;

// --> Wie bei Bank Avangard
      U     "MAL1S033".PCRead.Step.StPassive;
      R     "MAL1S033Par".Par.FlagMachine.WEGMESSUNG_0_FLAG;
      R     "MAL1S033Par".Par.FlagMachine.ImpulsNullstellung;
      R     "MAL1S033Par".Par.FlagMachine.CmdTurnFwdAfterLoading;
      R     "MAL1S033Par".Par.FlagMachine.CmdTurnRevAfterLoading;
      R     "MAL1S033Par".Par.FlagMachine.ImpulsNullstellungFP;
      R     "MAL1S033Par".Par.FlagMachine.CmdTurnFwdAfterTurning;
      R     "MAL1S033Par".Par.FlagMachine.CmdTurnRevAfterTurning;
      R     "MAL1S033Par".Par.FlagMachine.WEGMESSUNG_0;
      R     "MAL1S033Par".Par.FlagMachine.CmdTurnFwdAfterUnloading;
      R     "MAL1S033Par".Par.FlagMachine.CmdTurnRevAfterUnloading;
      R     "MAL1S033Par".Par.FlagMachine.NULL_INDEX_FP;
//
      U     "MAL1S033".PCRead.Step.StIdling;
      O     "MAL1S033".PCRead.Step.StPassive;
      SPBN  csn;
      L     0; // clear step number
      T     "MAL1S033Par".Par.ParIntMachine.ActualStep;
      T     "MAL1S033Par".StepAct.StepNumber;
csn:  NOP   0;

NETWORK
TITLE =Main0_End: Init flag
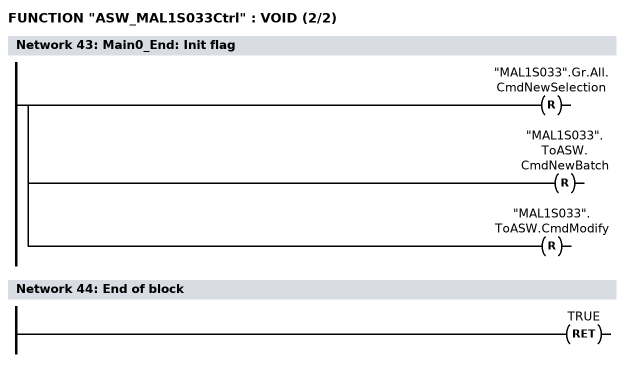

      SET   ;
      R     "MAL1S033".Gr.All.CmdNewSelection;
      R     "MAL1S033".ToASW.CmdNewBatch;
      R     "MAL1S033".ToASW.CmdModify;

NETWORK
TITLE =End of block

      BE    ;

END_FUNCTION

